PROGRAM PRG_MachineControl
VAR
    // =========================================================
    // TIMERS & TRIGGERS
    // =========================================================
	tonSys_Init           				: TON := (PT := T#8S);    // Initialization pulse timer
    tonSys_InitTimeout    				: TON := (PT := T#15S);   // Initialization timeout fault timer    : TON := (PT := T#15S);   // Initialization timeout fault timer
	tonTimeout_testing    				: TON := (PT := T#20S);   // Initialization timeout fault timer
    tonFirstAutoCycle     				: TON := (PT := T#500MS); // Auto cycle start settling timer
	tonStoppingDelay	  				: TON                   ; // Time to finalize process 
    tonSafety             				: TON := (PT := T#10S);   // Safety interlock debounce timer
	tonAutoCycleIdleTimeout 			: TON := (PT := T#2M);
	tonSimulation		  				: ARRAY[1..4] OF TON; //timer for simulations  
	rtKistlerResultDone   				: R_TRIG;
	rtPartPresentReject   				: R_TRIG;
    
    rtFirstAutoCycle      				: R_TRIG; // Detects entry into Auto Cycle
    fbResetTrigger        				: F_TRIG; // Detects HMI Reset button release
	tTwoHandReturnTimeout 				: TON := (PT := T#2S);
	tonAfterKistlerDelay  				: TON;
	
    eProcessCycleState : E_ProcessCycle_State := E_ProcessCycle_State.IDLE;
	
	tonGuideCylinderDelay 				: TON;
	tonGuideCylinderRetractDelay 		: TON;
	tGuideCylinderDelay   				: TIME := T#250MS;
	
	bFaultResetRequested 				: BOOL := FALSE;
	
    // =========================================================
    // PROCESS CYCLE CONTROL
    // =========================================================
	bStartProcessCondition 				: BOOL;   // OK to Start checklist condition flag
	bAutoCyclePermissive				: BOOL;
    bKistlerReady          				: BOOL;   // Press healthy and ready feedback flag
    i                      				: INT;    // Loop index counter
    sMachineMessage        				: STRING; // Diagnostics and status message string
	stKistlerInTelegram  				: ST_Kistler_TelegramIn;
	stKistlerOutTelegram 				: ST_Kistler_TelegramOut;
	
    bProcessCycleAllowed   		: BOOL;
    bAutoProcessAllowed    		: BOOL;
    bManualKistlerAllowed  		: BOOL;
	
	bAirInitialised     		: BOOL;
	bNestInitialised    		: BOOL;
	bKistlerInitialised 		: BOOL;
	bMachineInitialised 		: BOOL;
	
	bStopRequested 				: BOOL;
	bStopAllowed   				: BOOL;
	
	bRejectConfirmedForExchange : BOOL;
	bPendingOperatorResultPass  : BOOL;
	bPendingOperatorResultFail  : BOOL;
	
	// =================================================================
    // NEST TABLE INTERNAL CONTROL VARIABLES
    // =================================================================
	eNestState           			: E_NestState := E_NestState.IDLE;
	bSequenceToggle      			: BOOL := FALSE;                   // Toggle flag for manual bench testing
	eCurrentNestPos 	 			: E_NestPosition := E_NestPosition.UNKNOWN;
	eCompletedOperatorExchangeNest 	: E_NestPosition;
	
    // HMI PARAMETERS & SAFETY TIMERS
    rHmiTwoHandPresetTime 		: REAL := 250.0; // Time preset from HMI in milliseconds (e.g., 1500.0 ms = 1.5s)
    tTwoHandTargetTime    		: TIME;           // Converted time to be used by the PLC timer
    tTwoHandHoldTimer     		: TON;            // Timer to verify if operator held the buttons long enough
	
	// Timers for pneumatic steps control without sensors
	tSupportRetractDelay 		: TON;  // Time for elevator cylinder to retract down
	tRotatingTableDelay  		: TON;  // Simulated time for index table to complete rotation
	tPortB_ResetDelay    		: TON;  // Pulse time for Port B air relief / mechanism reset
	tSupportExtendDelay  		: TON;  // Time for elevator cylinder to extend back up
	
	eLastTestedNestPos 			: E_NestPosition := E_NestPosition.UNKNOWN;
	bNestNewPositionReady 		: BOOL;

	eOperatorExchangeState : E_OperatorExchangeState := E_OperatorExchangeState.Idle;

	bOperatorExchangeComplete 	 : BOOL;
	bOperatorIndexPermissive   	 : BOOL;
	
	//==========================================================
	//KISTLER COMMAND INTERFACE 
	//==========================================================
	stKistler_CMD          		: ST_Kistler_CMD;    // Commands sent to Kistler press
    stKistler_Status       		: ST_Kistler_Status; // Feedbacks read from Kistler press
	tonKistlerTareYDelay 		: TON;
	
	bKistlerResetPulse  		: BOOL;
    tonKistlerReset     		: TON;
	
	bKistlerRecoveryHomeRequest : BOOL;
	bNestRecoveryHomeRequest	: BOOL;
	uKistlerCurrentValueX 		: U_BytesToReal;
	uKistlerCurrentValueY 		: U_BytesToReal;
	
	// Maximum values recorded during the current Kistler test
	rKistlerCycleMaxForce    	: REAL := 0.0;
	rKistlerCycleMaxDistance 	: REAL := 0.0;

	

	//==========================================================
	//LEDS COMMAND INTERFACE 
	//==========================================================

    // Status memory for each individual LED mode
    eMode_LED_Start    			: E_LEDs_Mode := E_LEDs_Mode.OFF;
    eMode_LED_Reset    			: E_LEDs_Mode := E_LEDs_Mode.OFF;
	eMode_LED_Pass 	   			: E_LEDs_Mode := E_LEDs_Mode.OFF;
    eMode_LED_fail     			: E_LEDs_Mode := E_LEDs_Mode.OFF;
    // Hardware digital outputs mapped to the physical LEDs
    q_bLED_Start      AT%Q*    : BOOL; 
    q_bLED_Reset      AT%Q*    : BOOL;
	q_bLED_Pass       AT%Q*    : BOOL;
	q_bLED_Fail       AT%Q*    : BOOL;
    
	// =========================================================
    // PUCK LOCKER
    // =========================================================
	eKistlerNestPosition  		: E_NestPosition;
    eOperatorNestPosition 		: E_NestPosition;
	ePendingPuckDispositionNest : E_NestPosition := E_NestPosition.Unknown;

    iKistlerNestIndex     		: INT;
    iOperatorNestIndex    		: INT;
	
	bKistlerResultStored 		: BOOL;
	bPartRemovedConfirmedForExchange : BOOL;
	
    // =========================================================
    // PERSISTENT DATA & LOGGING
    // =========================================================
    //fbWritePersistent      : FB_WritePersistentData;
	bWriteTrigger         		: BOOL; // Test and simulation sequence trigger
	eCurrentState				: INT;
	
	// =========================================================
    // HMI COMMAND
    // =========================================================
	bHMIManualModeRequest 		: BOOL := FALSE;
	rtHMIManualModeRequest 		: R_TRIG;
	i_bHMIManualModeRequest		: INT;
	
	
	E_ProcessCycleState			: INT;
	IDLE						: INT;
END_VAR



// =========================================================
// 1. PRE-CONDITION LOGIC
// =========================================================
M_PreExecution();

// Generate Kistler commands based on current machine state
// Map Kistler EtherCAT telegram to PLC status structure
M_KistlerConfig_Output();

bStartProcessCondition :=
    GVL_MASTER.stMachineStatus.bSafety
    AND NOT GVL_MASTER.i_bButtonEmergencyStop
    AND NOT GVL_MASTER.stMachineStatus.bFault
    AND NOT stKistler_Status.bError
    AND stKistler_Status.bReady
    AND GVL_MASTER.stPuckLocker.bMachinePermissive;

 // Initialisation conditions
 
 	
	
    bAirInitialised := GVL_MASTER.bAirSupply_Ok;

    bNestInitialised :=
        (eNestState = E_NestState.IDLE)
        AND NOT GVL_MASTER.stNestTable.bNestInMotion
        AND GVL_MASTER.stNestTable.bNestReadySensor
        AND GVL_MASTER.stNestTable.bNestLockedSensor;

    bKistlerInitialised :=
         stKistler_Status.bInPosition
	      AND NOT stKistler_Status.bError;

    bMachineInitialised :=
        bAirInitialised
        AND bNestInitialised
        AND bKistlerInitialised;
		
	GVL_MASTER.bProcessBusy := 
	(eProcessCycleState <> E_ProcessCycle_State.WAIT_NEST_TESTING_READY 
	AND eProcessCycleState <> E_ProcessCycle_State.IDLE )
	
    OR (eNestState <> E_NestState.IDLE AND eNestState <> E_NestState.FAULT AND eNestState <> E_NestState.WAIT_OPERATOR_EXCHANGE)
    OR GVL_MASTER.stNestTable.bNestInMotion
    OR GVL_MASTER.stProcess.bKistlerCycleRequest
    OR GVL_MASTER.stProcess.bReleaseNestRotation
    OR stKistler_Status.bBusy
    OR NOT stKistler_Status.bInPosition
    OR GVL_MASTER.stNestTable.bSupportExtendRequest
    OR GVL_MASTER.stActuators.bGuideCylinderExtendRequest
	OR GVL_MASTER.stNestTable.bSupportExtended;
	
	

	
// =========================================================
// TIMEOUT
// =========================================================

	tonTimeout_testing (IN := GVL_MASTER.bProcessBusy);
	
	// Any process activity resets the accumulated timeout.
	tonAutoCycleIdleTimeout(
		IN :=
			GVL_MASTER.stMachineStatus.eMachineState =
				E_MachineState.SYSTEM_AUTO_CYCLE
			AND NOT GVL_MASTER.bProcessBusy
	);

// =========================================================
// GLOBAL FAULT DETECTION
// =========================================================
// Only technical Kistler errors shall put the machine in FAULT.
// Kistler NOK result is a rejected part, not a machine fault.
// =========================================================

//OR stKistler_Status.bError
IF (
    NOT GVL_MASTER.stMachineStatus.bSafety
    OR GVL_MASTER.i_bButtonEmergencyStop
)
AND GVL_MASTER.stMachineStatus.eMachineState <> E_MachineState.FAULT THEN

    GVL_MASTER.stMachineStatus.eMachineState := E_MachineState.FAULT;

END_IF;

//HMI Command Manual Mode

rtHMIManualModeRequest(CLK := GVL_HMI.i_bHMIManualModeRequest);

IF rtHMIManualModeRequest.Q AND GVL_Master.stMachineStatus.eMachineState = E_MachineState.SYSTEM_READY_TO_START THEN
    bHMIManualModeRequest := TRUE;
    GVL_HMI.i_bHMIManualModeRequest := FALSE;
ELSE
	bHMIManualModeRequest := FALSE;
    GVL_HMI.i_bHMIManualModeRequest := FALSE;
END_IF;


IF NOT GVL_MASTER.i_bButtonStop THEN
    bStopRequested := TRUE;
END_IF


	
IF GVL_MASTER.stMachineStatus.eMachineState <>
    E_MachineState.FAULT THEN

    bFaultResetRequested := FALSE;
END_IF;
// // =========================================================
// 2. MAIN STATE MACHINE (CASE)
// =========================================================


CASE GVL_Master.stMachineStatus.eMachineState OF


    E_MachineState.SYSTEM_POWER_UP:
	    GVL_Master.stMachineStatus.eMachineState := E_MachineState.STOPPING;
		M_ResetProcessCycle();
		
    E_MachineState.FAULT:
 		eMode_LED_Start := E_LEDs_Mode.OFF;
        eMode_LED_Reset := E_LEDs_Mode.FLASHING; // Reset button must flash
		eMode_LED_Fail := E_LEDs_Mode.ON;
		eMode_LED_PASS := E_LEDs_Mode.OFF;
		
		bHMIManualModeRequest := FALSE;
    	//M_ResetProcessCycle();
		
		 // Store the first reset request while TwinSAFE recovers.
		IF GVL_MASTER.i_bButtonReset THEN
			bFaultResetRequested := TRUE;
		END_IF;

		IF GVL_MASTER.stMachineStatus.bSafety
			AND NOT GVL_MASTER.i_bButtonEmergencyStop
		THEN
			bKistlerResetPulse := TRUE;
		END_IF;
	
	
		IF bKistlerResetPulse THEN
	
			IF M_ResetProcessCycle() THEN
	
				GVL_MASTER.stMachineStatus.eMachineState :=
					E_MachineState.STOPPING;
	
			END_IF;
	
		END_IF;

// 
//         IF  GVL_MASTER.stMachineStatus.bSafety AND NOT GVL_MASTER.i_bButtonEmergencyStop AND fbResetTrigger.Q THEN
//             GVL_Master.stMachineStatus.eMachineState := E_MachineState.STOPPING;
//         END_IF
		
	E_MachineState.STOPPING:
		eMode_LED_PASS := E_LEDs_Mode.OFF;
		eMode_LED_Fail := E_LEDs_Mode.OFF;
        rtFirstAutoCycle(CLK := FALSE);
        tonStoppingDelay(IN := GVL_Master.stMachineStatus.bStopping, PT := T#2S);
		bStopRequested := FALSE;
		IF tonStoppingDelay.Q THEN
			tonStoppingDelay(IN := FALSE);
        	GVL_Master.stMachineStatus.eMachineState := E_MachineState.STOPPED;
		END_IF
	   
	E_MachineState.STOPPED:
		eMode_LED_Reset := E_LEDs_Mode.FLASHING; // Start button must flash
        eMode_LED_Start := E_LEDs_Mode.OFF;
		eMode_LED_PASS := E_LEDs_Mode.OFF;
		eMode_LED_Fail := E_LEDs_Mode.OFF;
		M_ResetProcessCycle();

		IF fbResetTrigger.Q AND bStartProcessCondition THEN
            GVL_Master.stMachineStatus.eMachineState := E_MachineState.SYSTEM_INITIALISING;
			
        END_IF

		
	E_MachineState.SYSTEM_INITIALISING:
	
		tonSys_Init (IN := GVL_MASTER.stMachineStatus.bInitialising);
		tonSys_InitTimeout (IN := GVL_MASTER.stMachineStatus.bInitialising);
		eLastTestedNestPos := E_NestPosition.UNKNOWN;
		
		IF tonSys_Init.Q 
			AND GVL_IO.stSafety.bSafetyOK 
			AND bStartProcessCondition THEN
			
			IF NOT bKistlerInitialised THEN 
				
				 stKistler_Status.eKistlerState := E_KistlerState.HOMING;
    			 bKistlerRecoveryHomeRequest := TRUE;
				
			ELSIF   stKistler_Status.eKistlerState = E_KistlerState.READY THEN
   				GVL_MASTER.stMachineStatus.eMachineState := E_MachineState.SYSTEM_READY_TO_START;
			END_IF
			
		ELSIF tonSys_InitTimeout.Q THEN
			GVL_MASTER.stMachineStatus.eMachineState := E_MachineState.FAULT;
		
		ELSIF bStopRequested THEN
            GVL_Master.stMachineStatus.eMachineState := E_MachineState.STOPPING;
 		END_IF
// 		
	E_MachineState.SYSTEM_READY_TO_START:
	    
		eMode_LED_Start := E_LEDs_Mode.FLASHING; // Start button must flash
        eMode_LED_Reset := E_LEDs_Mode.OFF;
		eMode_LED_PASS := E_LEDs_Mode.OFF;
		eMode_LED_Fail := E_LEDs_Mode.OFF;
		
		IF bStopRequested THEN
            GVL_Master.stMachineStatus.eMachineState := E_MachineState.STOPPING;
	    		
        ELSIF bHMIManualModeRequest
   			AND GVL_MASTER.stMachineStatus.bSafety
   			AND NOT GVL_MASTER.i_bButtonEmergencyStop THEN
			//bHMIManualModeRequest := FALSE;
			GVL_Master.stMachineStatus.eMachineState := E_MachineState.MANUAL_MODE;
			
        ELSIF GVL_MASTER.i_bButtonStart
    			AND bStartProcessCondition
    			AND (stKistler_Status.eKistlerState = E_KistlerState.READY
        		OR stKistler_Status.eKistlerState = E_KistlerState.HOME_DONE) THEN
            		GVL_Master.stMachineStatus.eMachineState := E_MachineState.SYSTEM_AUTO_CYCLE;
			
		ELSIF  NOT GVL_IO.stSafety.bSafetyOK THEN
			GVL_Master.stMachineStatus.eMachineState := E_MachineState.FAULT;
        END_IF	
 
	E_MachineState.SYSTEM_AUTO_CYCLE:
	
		// Show the result of the processed part currently
		// waiting at the operator position.
		// -------------------------------------------------------------------------
		// Operator result indication.
		//
		// The LEDs must represent the stored result of the physical nest currently
		// available to the operator.
		//
		// Do not use bPendingOperatorResultPass / Fail here. Those variables are
		// latched for the operator-exchange state machine and may still represent
		// the previous exchange while the table is indexing.
		// -------------------------------------------------------------------------
		eMode_LED_PASS := E_LEDs_Mode.OFF;
		eMode_LED_Fail := E_LEDs_Mode.OFF;
		
		
		// The operator nest and its array index must be valid.
		IF eOperatorNestPosition <> E_NestPosition.Unknown THEN
		
			iOperatorNestIndex :=
				TO_INT(eOperatorNestPosition);
		
			IF (iOperatorNestIndex >= 1)
			   AND (iOperatorNestIndex <= 4) THEN
		
		
				// -------------------------------------------------------------
				// FAIL indication.
				//
				// Turn the red LED on as soon as the failed part arrives at the
				// operator position.
				//
				// Keep it on after the part is removed from the nest.
				//
				// Turn it off only after the reject sensor confirms that the
				// failed part was placed in the reject location.
				// -------------------------------------------------------------
				IF GVL_MASTER.astNestProcessResult[
						iOperatorNestIndex
				   ].bResultValid
				   AND GVL_MASTER.astNestProcessResult[
						iOperatorNestIndex
				   ].bFail
				   AND NOT bRejectConfirmedForExchange THEN
		
					eMode_LED_PASS := E_LEDs_Mode.OFF;
					eMode_LED_Fail := E_LEDs_Mode.ON;
		
		
				// -------------------------------------------------------------
				// PASS indication.
				//
				// Turn the green LED on as soon as the passed part arrives at
				// the operator position.
				//
				// Turn it off when the operator removes the part from the nest.
				// No puck condition is involved in the indication.
				// -------------------------------------------------------------
				ELSIF GVL_MASTER.astNestProcessResult[
							iOperatorNestIndex
					  ].bResultValid
					  AND GVL_MASTER.astNestProcessResult[
							iOperatorNestIndex
					  ].bPass
					  AND GVL_MASTER.stSensors.bPartPresent_NEST 
					  AND NOT bPartRemovedConfirmedForExchange THEN
		
					eMode_LED_PASS := E_LEDs_Mode.ON;
					eMode_LED_Fail := E_LEDs_Mode.OFF;
		
				END_IF
		
			END_IF
		
		END_IF
	
		rtFirstAutoCycle(CLK := TRUE);
		tonFirstAutoCycle(IN := rtFirstAutoCycle.Q);
	
		IF bStopRequested
			AND NOT GVL_MASTER.bProcessBusy THEN
	
			GVL_MASTER.stMachineStatus.eMachineState :=
				E_MachineState.STOPPING;
	
		ELSIF GVL_MASTER.stMachineStatus.bFault
			OR NOT bStartProcessCondition
			OR NOT GVL_IO.stSafety.bSafetyOK THEN
	
			GVL_MASTER.stMachineStatus.eMachineState :=
				E_MachineState.FAULT;
	
		ELSIF tonTimeout_testing.Q THEN
	
			GVL_MASTER.stMachineStatus.eMachineState :=
				E_MachineState.FAULT;
		ELSIF tonAutoCycleIdleTimeout.Q THEN

			GVL_MASTER.stMachineStatus.eMachineState :=
				E_MachineState.STOPPING;
	
		END_IF;
			
		
		
    E_MachineState.MANUAL_MODE:
		eMode_LED_Start := E_LEDs_Mode.OFF; // Start button must flash
        eMode_LED_Reset := E_LEDs_Mode.OFF;
		eMode_LED_PASS := E_LEDs_Mode.OFF;
		eMode_LED_Fail := E_LEDs_Mode.OFF;
		eLastTestedNestPos := E_NestPosition.UNKNOWN;
   		
		IF NOT GVL_MASTER.stMachineStatus.bSafety
		   OR GVL_MASTER.i_bButtonEmergencyStop THEN
		
			GVL_MASTER.stMachineStatus.eMachineState := E_MachineState.FAULT;
		
		ELSIF  bStopRequested 
			AND NOT GVL_MASTER.bProcessBusy THEN
			GVL_HMI.i_bHMIManualModeRequest				 := FALSE;
    		GVL_HMI.i_bHMIIndexerManualEnable 			 := FALSE;
    		GVL_HMI.i_bHMIKistlerManualEnable 			 := FALSE;
			GVL_MASTER.stMachineStatus.eMachineState := E_MachineState.STOPPING;
		
		END_IF

END_CASE

// =========================================================
// 3. GLOBAL FLAG MAPPING
// =========================================================
GVL_Master.stMachineStatus.bSystemPowerUp := (GVL_Master.stMachineStatus.eMachineState = E_MachineState.SYSTEM_POWER_UP);
GVL_Master.stMachineStatus.bInitialising  := (GVL_Master.stMachineStatus.eMachineState = E_MachineState.SYSTEM_INITIALISING);
GVL_Master.stMachineStatus.bStopped       := (GVL_Master.stMachineStatus.eMachineState = E_MachineState.STOPPED);
GVL_Master.stMachineStatus.bStopping      := (GVL_Master.stMachineStatus.eMachineState = E_MachineState.STOPPING);
GVL_Master.stMachineStatus.bAutoCycle     := (GVL_Master.stMachineStatus.eMachineState = E_MachineState.SYSTEM_AUTO_CYCLE);
GVL_Master.stMachineStatus.bFault         := (GVL_Master.stMachineStatus.eMachineState = E_MachineState.FAULT);
GVL_Master.stMachineStatus.bReadyToStart  := (GVL_Master.stMachineStatus.eMachineState = E_MachineState.SYSTEM_READY_TO_START);
GVL_Master.stMachineStatus.bManualMode    := (GVL_Master.stMachineStatus.eMachineState = E_MachineState.MANUAL_MODE);


// =========================================================
// 5. METHOD POST-EXECUTION ROUTINE
// =========================================================

// Generate base Kistler commands from machine state
M_KistlerControl(
    eCurrentState := GVL_MASTER.stMachineStatus.eMachineState);

// Coordinate Nest and Kistler process sequence
M_ProcessCycle();

// Update Puck locker permissives. 
M_UpdatePuckLockerPermissives();

// Kistler internal state machine may request movement/sequence
M_KistlerStateMachine(
    eCurrentState := GVL_MASTER.stMachineStatus.eMachineState);
	
M_SupportControl(
    bExtendRequest  := GVL_MASTER.stNestTable.bSupportExtendRequest,
    bRetractRequest := GVL_MASTER.stNestTable.bSupportRetractRequest
);

M_GuideCylinderControl(
    bExtendRequest := GVL_MASTER.stActuators.bGuideCylinderExtendRequest
);

M_KistlerConfig_Input();

// Update machine status from Kistler status
M_StatusMapping();

M_LEDsButtons();
M_NestTableControl();

METHOD PRIVATE M_ClearCompletedOperatorNestResult
VAR
	iCompletedNestIndex : INT;
END_VAR
// The nest associated with the completed exchange must be known.
IF eCompletedOperatorExchangeNest = E_NestPosition.Unknown THEN
    RETURN;
END_IF

iCompletedNestIndex := TO_INT(eCompletedOperatorExchangeNest);

IF (iCompletedNestIndex < 1) OR (iCompletedNestIndex > 4) THEN
    RETURN;
END_IF


// Clear only after the complete operator disposition has finished.
GVL_MASTER.astNestProcessResult[iCompletedNestIndex].bResultValid := FALSE;
GVL_MASTER.astNestProcessResult[iCompletedNestIndex].bPass := FALSE;
GVL_MASTER.astNestProcessResult[iCompletedNestIndex].bFail := FALSE;
GVL_MASTER.astNestProcessResult[iCompletedNestIndex].bDispositionSent := FALSE;

eCompletedOperatorExchangeNest := E_NestPosition.Unknown;
END_METHOD

METHOD PRIVATE M_ClearRemovedOperatorNestResult
VAR
	iOperatorNestIndex : INT;
END_VAR
// The operator nest must be known.
IF eOperatorNestPosition = E_NestPosition.Unknown THEN
    RETURN;
END_IF


// E_NestPosition corresponds directly to indexes 1..4.
iOperatorNestIndex := TO_INT(eOperatorNestPosition);

IF (iOperatorNestIndex < 1) OR (iOperatorNestIndex > 4) THEN
    RETURN;
END_IF


// Clear the stored result only when:
//
// 1. The result was already delivered to the Puck Locker.
// 2. The processed part was physically removed from the operator nest.
IF GVL_MASTER.astNestProcessResult[iOperatorNestIndex].bDispositionSent AND GVL_MASTER.astNestTracking[iOperatorNestIndex].bPartRemovedPulse THEN

    GVL_MASTER.astNestProcessResult[iOperatorNestIndex].bResultValid := FALSE;

    GVL_MASTER.astNestProcessResult[iOperatorNestIndex].bPass := FALSE;

    GVL_MASTER.astNestProcessResult[iOperatorNestIndex].bFail := FALSE;

    GVL_MASTER.astNestProcessResult[iOperatorNestIndex].bDispositionSent := FALSE;

END_IF;
END_METHOD

METHOD PRIVATE M_ConfirmPuckLockerDisposition
VAR
	iDispositionNestIndex : INT;
END_VAR
// No disposition is waiting for confirmation.
IF ePendingPuckDispositionNest = E_NestPosition.Unknown THEN
    RETURN;
END_IF


// The Puck Locker has not yet consumed the request.
IF NOT GVL_MASTER.stPuckLocker.bDispositionHandled THEN
    RETURN;
END_IF


// E_NestPosition values correspond directly to indexes 1..4.
iDispositionNestIndex :=
    ePendingPuckDispositionNest;

IF (iDispositionNestIndex < 1) OR (iDispositionNestIndex > 4) THEN

    // Prevent the handshake from remaining blocked by an invalid position.
    ePendingPuckDispositionNest :=
        E_NestPosition.Unknown;
    RETURN;
END_IF


// Mark the result as successfully delivered to the Puck Locker.
GVL_MASTER.astNestProcessResult[iDispositionNestIndex].bDispositionSent := TRUE;


// Release the local handshake.
ePendingPuckDispositionNest := E_NestPosition.Unknown;
END_METHOD

METHOD M_GetCurrentPosition : E_NestPosition
VAR_INST
	iBinaryValue : BYTE;
END_VAR
// 1. Pack the 3 boolean sensors into a single numeric value (Byte) to simplify binary calculation
// Sensor_3 (Bit 2) | Sensor_2 (Bit 1) | Sensor_1 (Bit 0)
iBinaryValue.0 := GVL_MASTER.stNestTable.bNestPos_1_Sensor;
iBinaryValue.1 := GVL_MASTER.stNestTable.bNestPos_2_Sensor;
iBinaryValue.2 := GVL_MASTER.stNestTable.bNestPos_3_Sensor;

// 2. Evaluate the resulting decimal value from the binary combination and return the matching ENUM
CASE iBinaryValue OF
    1: M_GetCurrentPosition := E_NestPosition.POSITION_1; // Binary 001
    2: M_GetCurrentPosition := E_NestPosition.POSITION_2; // Binary 010
    3: M_GetCurrentPosition := E_NestPosition.POSITION_3; // Binary 011
    4: M_GetCurrentPosition := E_NestPosition.POSITION_4; // Binary 100
ELSE
    // Default fallback: If 000 or any unmapped pattern occurs (e.g., 111), the table might be misaligned or in motion
    M_GetCurrentPosition := E_NestPosition.UNKNOWN; 
END_CASE


CASE eCurrentNestPos OF
    E_NestPosition.POSITION_1:
        GVL_HMI.iNestRotationAngle      := 0;
		GVL_HMI.iNestPositionTesting    :=1;

    E_NestPosition.POSITION_2:
        GVL_HMI.iNestRotationAngle 		:= 90;
		GVL_HMI.iNestPositionTesting    :=2;
		
    E_NestPosition.POSITION_3:
        GVL_HMI.iNestRotationAngle 		:= 180;
	    GVL_HMI.iNestPositionTesting    :=3;
		
    E_NestPosition.POSITION_4:
        GVL_HMI.iNestRotationAngle 		:= 270;
		GVL_HMI.iNestPositionTesting    :=4;

ELSE
    GVL_HMI.iNestRotationAngle      := 0;
	GVL_HMI.iNestPositionTesting    := 0;
END_CASE
END_METHOD

METHOD PRIVATE M_GuideCylinderControl
VAR_INPUT
    bExtendRequest : BOOL;
END_VAR
// =================================================================
// GUIDE CYLINDER CONTROL
// =================================================================
// This method is responsible only for the Guide Cylinder output.
// It does not decide Auto Cycle or Manual Mode.
// The request must come from the Kistler state machine.
//
// Single-solenoid pneumatic cylinder:
// TRUE  -> Extend guide cylinder.
// FALSE -> Retract guide cylinder automatically.

GVL_MASTER.stActuators.qGuideCylinder := bExtendRequest;
END_METHOD

METHOD PRIVATE M_HMIKistlerResult : BOOL
VAR_INPUT
    eNestPosition : E_NestPosition;
    bPartOK       : BOOL;
    bPartNOK      : BOOL;
    rForce        : REAL;
    rDistance     : REAL;
	bResetValues  : BOOL;
END_VAR

VAR
    iNestIndex : INT;
END_VAR


M_HMIKistlerResult := FALSE;


// =========================================================
// CONVERT NEST POSITION TO ARRAY INDEX
// =========================================================

CASE eNestPosition OF

    E_NestPosition.Position_1:
        iNestIndex := 1;

    E_NestPosition.Position_2:
        iNestIndex := 2;

    E_NestPosition.Position_3:
        iNestIndex := 3;

    E_NestPosition.Position_4:
        iNestIndex := 4;

ELSE
    RETURN;

END_CASE;


// =========================================================
// RESET VALUES BEFORE A NEW TEST
// =========================================================

IF bResetValues THEN

    GVL_HMI.aKistlerNestResult[iNestIndex].rForce := 0.0;
    GVL_HMI.aKistlerNestResult[iNestIndex].rDistance := 0.0;

    GVL_HMI.aKistlerNestResult[iNestIndex].eResult :=
        E_HMIKistlerResult.NONE;

    M_HMIKistlerResult := TRUE;
    RETURN;

END_IF;


// =========================================================
// STORE MAXIMUM TEST VALUES
// =========================================================

IF ABS(rForce) >
   ABS(GVL_HMI.aKistlerNestResult[iNestIndex].rForce) THEN

    GVL_HMI.aKistlerNestResult[iNestIndex].rForce :=
        rForce;

END_IF;


IF ABS(rDistance) >
   ABS(GVL_HMI.aKistlerNestResult[iNestIndex].rDistance) THEN

    GVL_HMI.aKistlerNestResult[iNestIndex].rDistance :=
        rDistance;

END_IF;


// =========================================================
// STORE FINAL RESULT
// =========================================================

IF bPartOK THEN

    GVL_HMI.aKistlerNestResult[iNestIndex].eResult :=
        E_HMIKistlerResult.PASS;

ELSIF bPartNOK THEN

    GVL_HMI.aKistlerNestResult[iNestIndex].eResult :=
        E_HMIKistlerResult.FAIL;

END_IF;


M_HMIKistlerResult := TRUE;
END_METHOD

METHOD M_IsNestEnabled :BOOL
VAR_INPUT
	   eNestPos : E_NestPosition;
END_VAR
CASE eNestPos OF

    E_NestPosition.Position_1:
        M_IsNestEnabled := GVL_HMI.aNestEnabled[1];

    E_NestPosition.Position_2:
        M_IsNestEnabled := GVL_HMI.aNestEnabled[2];

    E_NestPosition.Position_3:
        M_IsNestEnabled := GVL_HMI.aNestEnabled[3];

    E_NestPosition.Position_4:
        M_IsNestEnabled := GVL_HMI.aNestEnabled[4];

ELSE

    M_IsNestEnabled := FALSE;

END_CASE;
END_METHOD

METHOD PRIVATE M_KistlerCommandMapping : BOOL
VAR
    i : INT;
END_VAR

// =================================================================================
// PLC -> KISTLER COMMAND MAPPING
// =================================================================================
// Clear command telegram
FOR i := 0 TO 199 DO
    GVL_KISTLER_IO.aKistlerOut[i] := 0;
END_FOR

// Enable maXYmos access and automatic mode
IF stKistler_CMD.bEnable THEN
    GVL_KISTLER_IO.aKistlerOut[1].3 := TRUE; // Access
    GVL_KISTLER_IO.aKistlerOut[1].4 := TRUE; // Auto
    GVL_KISTLER_IO.aKistlerOut[9].0 := TRUE; // Drive_Enable
END_IF

// Reset / acknowledge maXYmos faults/statistics
IF stKistler_CMD.bReset THEN
    GVL_KISTLER_IO.aKistlerOut[1].0 := TRUE; // Ack_Admin_Glob
    GVL_KISTLER_IO.aKistlerOut[1].1 := TRUE; // Ack_Admin
    GVL_KISTLER_IO.aKistlerOut[1].5 := TRUE; // Start_Reset
END_IF

// Abort / external sequence stop
IF stKistler_CMD.bAbort THEN
    GVL_KISTLER_IO.aKistlerOut[10].3 := TRUE; // Seq_Ext_Stop
END_IF

// Force Measurement Program 1 for first commissioning test
GVL_KISTLER_IO.aKistlerOut[2].0 := TRUE; // MP_01




M_KistlerCommandMapping := TRUE;
END_METHOD

METHOD PRIVATE M_KistlerConfig_Input : BOOL
VAR
    i : INT;
END_VAR
// =================================================================================
// KISTLER CONFIG INPUT
// PLC -> maXYmos NC input/control telegram
// =================================================================================
// Source:
//     stKistler_CMD
//
// Internal telegram:
//     stKistlerInTelegram
//
// Destination:
//     GVL_KISTLER_IO.aKistlerOut[]
// =================================================================================


// =================================================================================
// CLEAR OUTPUT TELEGRAM
// =================================================================================

FOR i := 0 TO 199 DO
    GVL_KISTLER_IO.aKistlerOut[i] := 0;
END_FOR



// =================================================================================
// HIGH LEVEL COMMANDS -> KISTLER INPUT TELEGRAM STRUCT
// =================================================================================

// -----------------------------------------------------------------------------
// Byte 0 - Measurement commands
// NOTE:
// Byte 0.0 = Measurement START.
// This is NOT the same as Start Sequence.
// Start Sequence is controlled by Byte 9.1 = Run Sequence.
// -----------------------------------------------------------------------------

stKistlerInTelegram.bStart := stKistler_CMD.bStart;
stKistlerInTelegram.bTareY := stKistler_CMD.bTareY;


// -----------------------------------------------------------------------------
// Byte 1 - General control
// -----------------------------------------------------------------------------

stKistlerInTelegram.bAckAdminGlobal := stKistler_CMD.bReset;
stKistlerInTelegram.bAckAdmin       := stKistler_CMD.bReset;
//stKistlerInTelegram.bStatReset      := stKistler_CMD.bReset;
stKistlerInTelegram.bAccess         := stKistler_CMD.bEnable;
stKistlerInTelegram.bAuto           := stKistler_CMD.bEnable;
stKistlerInTelegram.bStatReset       := FALSE;

// -----------------------------------------------------------------------------
// Byte 2 - Measurement program selection
// Byte 2 bits 0..6 = MP selection
// 0 = MP_000
// -----------------------------------------------------------------------------

stKistlerInTelegram.byMeasurementProgram := 0;


// -----------------------------------------------------------------------------
// Byte 9 - Drive / sequence commands
// -----------------------------------------------------------------------------

stKistlerInTelegram.bDriveEnable      := stKistler_CMD.bEnable;
stKistlerInTelegram.bRunSequence      := stKistler_CMD.bRunSequence;
stKistlerInTelegram.bDriveToHomePos   := stKistler_CMD.bDriveToHome;
stKistlerInTelegram.bDriveToRefPos    := stKistler_CMD.bDriveToRef;
stKistlerInTelegram.bContinueFromWait := stKistler_CMD.bContinueFromWait;


// -----------------------------------------------------------------------------
// Byte 10 - External sequence stop request
// -----------------------------------------------------------------------------

stKistlerInTelegram.bSeqExtStopReq := stKistler_CMD.bAbort;


// -----------------------------------------------------------------------------
// Byte 12 - Current sequence selection
// 00 = Main sequence
// 01 = Sub1
// 10 = Sub2
// 11 = Sub3
//
// For current commissioning, always use Main Sequence.
// -----------------------------------------------------------------------------

stKistlerInTelegram.bCurrentSequence0 := FALSE;
stKistlerInTelegram.bCurrentSequence1 := FALSE;


// =================================================================================
// KISTLER INPUT TELEGRAM STRUCT -> OUTPUT BYTES
// =================================================================================

IF stKistlerInTelegram.bDriveToHomePos THEN

    stKistlerInTelegram.bDriveToRefPos := FALSE;
    stKistlerInTelegram.bRunSequence   := FALSE;

ELSIF stKistlerInTelegram.bDriveToRefPos THEN

    stKistlerInTelegram.bDriveToHomePos := FALSE;
    stKistlerInTelegram.bRunSequence    := FALSE;

ELSIF stKistlerInTelegram.bRunSequence THEN

    stKistlerInTelegram.bDriveToHomePos := FALSE;
    stKistlerInTelegram.bDriveToRefPos  := FALSE;

END_IF
// -----------------------------------------------------------------------------
// -----------------------------------------------------------------------------
// Byte 0 - Measurement commands
// Bit 0 = Measurement Start
// Bit 1 = Tare Y
// -----------------------------------------------------------------------------
// -----------------------------------------------------------------------------

GVL_KISTLER_IO.aKistlerOut[0].0 := stKistlerInTelegram.bStart;
GVL_KISTLER_IO.aKistlerOut[0].1 := stKistlerInTelegram.bTareY;


// -----------------------------------------------------------------------------
// Byte 1 - General control
// -----------------------------------------------------------------------------

GVL_KISTLER_IO.aKistlerOut[1].0 := stKistlerInTelegram.bAckAdminGlobal;
GVL_KISTLER_IO.aKistlerOut[1].1 := stKistlerInTelegram.bAckAdmin;
GVL_KISTLER_IO.aKistlerOut[1].3 := stKistlerInTelegram.bAccess;
GVL_KISTLER_IO.aKistlerOut[1].4 := stKistlerInTelegram.bAuto;
GVL_KISTLER_IO.aKistlerOut[1].5 := stKistlerInTelegram.bStatReset;


// -----------------------------------------------------------------------------
// Byte 2 - Measurement program selection
// -----------------------------------------------------------------------------

GVL_KISTLER_IO.aKistlerOut[2] := stKistlerInTelegram.byMeasurementProgram;


// -----------------------------------------------------------------------------
// Byte 9 - Drive / sequence commands
// Bit 0 = Drive Enable
// Bit 1 = Run Sequence / Start Sequence
// Bit 2 = Drive To Home Position
// Bit 3 = Drive To Reference Position
// Bit 6 = Continue From Wait
// -----------------------------------------------------------------------------

GVL_KISTLER_IO.aKistlerOut[9].0 := stKistlerInTelegram.bDriveEnable;
GVL_KISTLER_IO.aKistlerOut[9].1 := stKistlerInTelegram.bRunSequence;
GVL_KISTLER_IO.aKistlerOut[9].2 := stKistlerInTelegram.bDriveToHomePos;
GVL_KISTLER_IO.aKistlerOut[9].3 := stKistlerInTelegram.bDriveToRefPos;
GVL_KISTLER_IO.aKistlerOut[9].6 := stKistlerInTelegram.bContinueFromWait;


// -----------------------------------------------------------------------------
// Byte 10 - External sequence stop request
// Bit 3 = Sequence External Stop Request
// -----------------------------------------------------------------------------

GVL_KISTLER_IO.aKistlerOut[10].3 := stKistlerInTelegram.bSeqExtStopReq;


// -----------------------------------------------------------------------------
// Byte 12 - Current sequence selection
// 00 = Main sequence
// 01 = Sub1
// 10 = Sub2
// 11 = Sub3
// -----------------------------------------------------------------------------

GVL_KISTLER_IO.aKistlerOut[12].0 := stKistlerInTelegram.bCurrentSequence0;
GVL_KISTLER_IO.aKistlerOut[12].1 := stKistlerInTelegram.bCurrentSequence1;


// =================================================================================
// METHOD EXECUTION FEEDBACK
// =================================================================================

M_KistlerConfig_Input := TRUE;
END_METHOD

METHOD PRIVATE M_KistlerConfig_Output : BOOL
VAR_INPUT
END_VAR
// =================================================================================
// INPUT BYTES -> KISTLER OUTPUT TELEGRAM STRUCT
// =================================================================================
// Byte 0 - Mirrored measurement commands
stKistlerOutTelegram.bMirrorStart             := GVL_KISTLER_IO.aKistlerIn[0].0;
stKistlerOutTelegram.bMirrorTareY             := GVL_KISTLER_IO.aKistlerIn[0].1;
stKistlerOutTelegram.bMirrorZeroX             := GVL_KISTLER_IO.aKistlerIn[0].2;
stKistlerOutTelegram.bMirrorSensorTestX       := GVL_KISTLER_IO.aKistlerIn[0].3;
stKistlerOutTelegram.bMirrorSensorTestY       := GVL_KISTLER_IO.aKistlerIn[0].4;
stKistlerOutTelegram.bMirrorMasterMeasurement := GVL_KISTLER_IO.aKistlerIn[0].6;
stKistlerOutTelegram.bMirrorIncZero           := GVL_KISTLER_IO.aKistlerIn[0].7;

// Byte 1 - Mirrored general control
stKistlerOutTelegram.bMirrorAckAdminGlobal := GVL_KISTLER_IO.aKistlerIn[1].0;
stKistlerOutTelegram.bMirrorAckAdmin       := GVL_KISTLER_IO.aKistlerIn[1].1;
stKistlerOutTelegram.bMirrorAccess         := GVL_KISTLER_IO.aKistlerIn[1].3;
stKistlerOutTelegram.bMirrorAuto           := GVL_KISTLER_IO.aKistlerIn[1].4;
stKistlerOutTelegram.bMirrorStatReset      := GVL_KISTLER_IO.aKistlerIn[1].5;
stKistlerOutTelegram.bMirrorStatDisable    := GVL_KISTLER_IO.aKistlerIn[1].6;
stKistlerOutTelegram.bMirrorTareExtendedY  := GVL_KISTLER_IO.aKistlerIn[1].7;

// Byte 2 - Mirrored MP
stKistlerOutTelegram.byMirrorMeasurementProgram := GVL_KISTLER_IO.aKistlerIn[2];

// Byte 3 - Mirrored special commands / reserved
stKistlerOutTelegram.bMirrorResetSNGenerator := GVL_KISTLER_IO.aKistlerIn[3].1;
stKistlerOutTelegram.bMirrorBrakeTestActive  := GVL_KISTLER_IO.aKistlerIn[3].5;
stKistlerOutTelegram.bMirrorExportPVTStatus  := GVL_KISTLER_IO.aKistlerIn[3].6;

// Byte 5 - Reserved
stKistlerOutTelegram.byReserved05 := GVL_KISTLER_IO.aKistlerIn[5];

// Byte 4 - Mirrored configurable inputs
stKistlerOutTelegram.bMirrorInput00 := GVL_KISTLER_IO.aKistlerIn[4].0;
stKistlerOutTelegram.bMirrorInput01 := GVL_KISTLER_IO.aKistlerIn[4].1;
stKistlerOutTelegram.bMirrorInput02 := GVL_KISTLER_IO.aKistlerIn[4].2;
stKistlerOutTelegram.bMirrorInput03 := GVL_KISTLER_IO.aKistlerIn[4].3;
stKistlerOutTelegram.bMirrorInput04 := GVL_KISTLER_IO.aKistlerIn[4].4;
stKistlerOutTelegram.bMirrorInput05 := GVL_KISTLER_IO.aKistlerIn[4].5;
stKistlerOutTelegram.bMirrorInput06 := GVL_KISTLER_IO.aKistlerIn[4].6;
stKistlerOutTelegram.bMirrorInput07 := GVL_KISTLER_IO.aKistlerIn[4].7;

// Byte 6 - General status
stKistlerOutTelegram.bReady    := GVL_KISTLER_IO.aKistlerIn[6].0;
stKistlerOutTelegram.bOkTotal  := GVL_KISTLER_IO.aKistlerIn[6].1;
stKistlerOutTelegram.bNokTotal := GVL_KISTLER_IO.aKistlerIn[6].2;
stKistlerOutTelegram.bWarning  := GVL_KISTLER_IO.aKistlerIn[6].6;
stKistlerOutTelegram.bAlarm    := GVL_KISTLER_IO.aKistlerIn[6].7;

// Byte 9 - Mirrored commands / sequence request
stKistlerOutTelegram.bMirrorDriveEnable    := GVL_KISTLER_IO.aKistlerIn[9].0;
stKistlerOutTelegram.bMirrorRunSequence    := GVL_KISTLER_IO.aKistlerIn[9].1;
stKistlerOutTelegram.bMirrorDriveToHomePos := GVL_KISTLER_IO.aKistlerIn[9].2;
stKistlerOutTelegram.bMirrorDriveToRefPos  := GVL_KISTLER_IO.aKistlerIn[9].3;
stKistlerOutTelegram.bWaitRequest          := GVL_KISTLER_IO.aKistlerIn[9].6;

// Byte 10 - Sequence / drive status
stKistlerOutTelegram.bSequenceStopped := GVL_KISTLER_IO.aKistlerIn[10].0;
stKistlerOutTelegram.bSequenceEnd     := GVL_KISTLER_IO.aKistlerIn[10].1;
//stKistlerOutTelegram.bSequenceError   := GVL_KISTLER_IO.aKistlerIn[10].4;
stKistlerOutTelegram.bSequenceError   := FALSE;
stKistlerOutTelegram.bDriveEnabled    := GVL_KISTLER_IO.aKistlerIn[10].5; // olhar essa 
stKistlerOutTelegram.bHomePosReached  := GVL_KISTLER_IO.aKistlerIn[10].6;
stKistlerOutTelegram.bRefPosReached   := GVL_KISTLER_IO.aKistlerIn[10].7;

// Byte 11 - Servo / safety status
stKistlerOutTelegram.bStandStill       := GVL_KISTLER_IO.aKistlerIn[11].0;
stKistlerOutTelegram.bServoWarning     := GVL_KISTLER_IO.aKistlerIn[11].2;
//stKistlerOutTelegram.bServoError       := GVL_KISTLER_IO.aKistlerIn[11].3;
stKistlerOutTelegram.bServoError       := FALSE;
stKistlerOutTelegram.bSMES_STO         := GVL_KISTLER_IO.aKistlerIn[11].4;
stKistlerOutTelegram.bSMST             := GVL_KISTLER_IO.aKistlerIn[11].5;
stKistlerOutTelegram.bSMM              := GVL_KISTLER_IO.aKistlerIn[11].6;
stKistlerOutTelegram.bUserModeActive   := GVL_KISTLER_IO.aKistlerIn[11].7;

// Byte 19 - Communication status
//stKistlerOutTelegram.bTransmissionFault := GVL_KISTLER_IO.aKistlerIn[19].0;
stKistlerOutTelegram.bTransmissionFault := FALSE;
stKistlerOutTelegram.bAck               := GVL_KISTLER_IO.aKistlerIn[19].1;
stKistlerOutTelegram.bDeviceAvailable   := GVL_KISTLER_IO.aKistlerIn[19].2;

// =================================================================================
// KISTLER OUTPUT TELEGRAM STRUCT -> INTERNAL STATUS
// =================================================================================

// =================================================================================
// INTERNAL STATUS
// =================================================================================

// Kistler is ready from communication/device point of view.
// This does not mean machine is allowed to run.
stKistler_Status.bReady :=
    stKistlerOutTelegram.bDeviceAvailable
    AND NOT stKistlerOutTelegram.bServoError
    AND NOT stKistlerOutTelegram.bTransmissionFault;


// Sequence is running.
// MirrorRunSequence confirms command accepted, and SequenceEnd is still false.
stKistler_Status.bBusy :=
    stKistlerOutTelegram.bMirrorRunSequence
    AND NOT stKistlerOutTelegram.bSequenceEnd
    AND NOT stKistlerOutTelegram.bSequenceStopped;


// Sequence finished, regardless of OK or NOK result.
stKistler_Status.bDone :=
    stKistlerOutTelegram.bSequenceEnd;


// Part result OK.
stKistler_Status.bPartOK :=
    stKistlerOutTelegram.bSequenceEnd
    AND stKistlerOutTelegram.bOkTotal;


// Part result NOK / rejected part.
// Important: this is NOT a technical error.
stKistler_Status.bPartNOK :=
    stKistlerOutTelegram.bSequenceEnd
    AND stKistlerOutTelegram.bNokTotal;


// Technical error only.
// NOK result must not be included here.
// stKistler_Status.bError :=
//     stKistlerOutTelegram.bServoError
//     OR stKistlerOutTelegram.bTransmissionFault
//     OR stKistlerOutTelegram.bSequenceError;


// Position status
stKistler_Status.bInPosition :=
    stKistlerOutTelegram.bHomePosReached;



// =================================================================================
// BYTES 20..23 - CURRENT X VALUE
// X = DISTANCE / DISPLACEMENT / TRAVEL
// =================================================================================

uKistlerCurrentValueX.aBytes[0] := GVL_KISTLER_IO.aKistlerIn[20];
uKistlerCurrentValueX.aBytes[1] := GVL_KISTLER_IO.aKistlerIn[21];
uKistlerCurrentValueX.aBytes[2] := GVL_KISTLER_IO.aKistlerIn[22];
uKistlerCurrentValueX.aBytes[3] := GVL_KISTLER_IO.aKistlerIn[23];

stKistlerOutTelegram.rCurrentValueX :=
    uKistlerCurrentValueX.rValue;


// =================================================================================
// BYTES 24..27 - CURRENT Y VALUE
// Y = FORCE
// =================================================================================

uKistlerCurrentValueY.aBytes[0] := GVL_KISTLER_IO.aKistlerIn[24];
uKistlerCurrentValueY.aBytes[1] := GVL_KISTLER_IO.aKistlerIn[25];
uKistlerCurrentValueY.aBytes[2] := GVL_KISTLER_IO.aKistlerIn[26];
uKistlerCurrentValueY.aBytes[3] := GVL_KISTLER_IO.aKistlerIn[27];

stKistlerOutTelegram.rCurrentValueY :=
    uKistlerCurrentValueY.rValue;
	
	
	// =================================================================================
// MAP LIVE VALUES TO INTERNAL KISTLER STATUS
// =================================================================================

stKistler_Status.rLiveDistance :=
    stKistlerOutTelegram.rCurrentValueX;

stKistler_Status.rLiveForce :=
    stKistlerOutTelegram.rCurrentValueY;


// =================================================================================
// OPTIONAL LIVE VALUES FOR HMI
// =================================================================================

GVL_HMI.rKistlerLiveDistance :=
    stKistler_Status.rLiveDistance;

GVL_HMI.rKistlerLiveForce :=
    stKistler_Status.rLiveForce;
// =================================================================================
// METHOD EXECUTION FEEDBACK
// =================================================================================

M_KistlerConfig_Output := TRUE;
END_METHOD

METHOD PRIVATE M_KistlerControl : BOOL
VAR_INPUT
    eCurrentState : E_MachineState;
END_VAR

VAR
    bKistlerSafetyEnableOK : BOOL;
END_VAR


// =========================================================
// RESET BUTTON DETECTION
// =========================================================

// F_TRIG generates the event when the reset button is released
fbResetTrigger(
    CLK := GVL_MASTER.i_bButtonReset
);


// Perform the complete process reset only in allowed states
IF fbResetTrigger.Q
    AND eCurrentState <> E_MachineState.SYSTEM_AUTO_CYCLE
    AND eCurrentState <> E_MachineState.SYSTEM_READY_TO_START
THEN

    M_ResetProcessCycle();

END_IF;


// =========================================================
// KISTLER RESET / ALARM ACKNOWLEDGEMENT PULSE
// =========================================================

// bKistlerResetPulse is set by M_ResetProcessCycle()
tonKistlerReset(
    IN := bKistlerResetPulse,
    PT := T#500MS
);

// This is the command that is actually sent to the Kistler
stKistler_CMD.bReset := bKistlerResetPulse;


// End the pulse after 500 ms
IF tonKistlerReset.Q THEN

    bKistlerResetPulse := FALSE;

END_IF;


// =========================================================
// ABORT
// =========================================================

// Keep abort active while the machine is faulted
stKistler_CMD.bAbort :=
    eCurrentState = E_MachineState.FAULT;


// =========================================================
// ENABLE
// =========================================================

stKistler_CMD.bEnable :=
    GVL_MASTER.stMachineStatus.bSafety
    AND GVL_KISTLER_IO.bKistlerSafetyEnableOK
    AND NOT GVL_MASTER.i_bButtonEmergencyStop
    AND NOT GVL_MASTER.stMachineStatus.bFault
    AND
    (
        eCurrentState = E_MachineState.SYSTEM_INITIALISING
        OR eCurrentState = E_MachineState.SYSTEM_READY_TO_START
        OR eCurrentState = E_MachineState.SYSTEM_AUTO_CYCLE
        OR eCurrentState = E_MachineState.STOPPING
        OR
        (
            eCurrentState = E_MachineState.MANUAL_MODE
            AND GVL_HMI.i_bHMIKistlerManualEnable
        )
    );


// =========================================================
// MANUAL MODE
// =========================================================

stKistler_CMD.bManualMode :=
    eCurrentState = E_MachineState.MANUAL_MODE
    AND GVL_HMI.i_bHMIKistlerManualEnable;


// =========================================================
// MOTION / SEQUENCE COMMAND DEFAULTS
// =========================================================

// M_KistlerStateMachine(), called later in the PLC cycle,
// may activate these commands when required.

stKistler_CMD.bStart            := FALSE;
stKistler_CMD.bRunSequence      := FALSE;
stKistler_CMD.bDriveToHome      := FALSE;
stKistler_CMD.bDriveToRef       := FALSE;
stKistler_CMD.bContinueFromWait := FALSE;
stKistler_CMD.bTareY            := FALSE;


// =========================================================
// METHOD EXECUTION FEEDBACK
// =========================================================

M_KistlerControl := TRUE;
END_METHOD

METHOD PRIVATE M_KistlerStateMachine : BOOL

VAR_INPUT
    eCurrentState : E_MachineState;

END_VAR

VAR
    bKistlerEnableAllowed    : BOOL;
    bKistlerAutoCycleAllowed : BOOL;
    bKistlerManualAllowed    : BOOL;
    bKistlerSequenceAllowed  : BOOL;
	

	
	
	Teste 			: BOOL :=TRUE;
END_VAR

VAR_INST
    rTrigTwoHands : R_TRIG; // Edge trigger to detect single press of the two-hand safety signal

END_VAR
// =================================================================================
// KISTLER STATE MACHINE
// maXYmos NC logical sequence control
// =================================================================================
// Input:
//     eCurrentState
//     stKistlerOutTelegram
//     stKistler_Status
//
// Output:
//     stKistler_CMD
// =================================================================================


// =================================================================================
// KISTLER OPERATION MODE PERMISSIVES
// =================================================================================

// Kistler may be enabled and stay READY in Ready To Start.
// It may also be enabled during Auto Cycle.
// In Manual Mode, it may be enabled only when the HMI manual enable is active.
bKistlerEnableAllowed :=
    (eCurrentState = E_MachineState.SYSTEM_READY_TO_START)
    OR (eCurrentState = E_MachineState.SYSTEM_AUTO_CYCLE)
	OR (eCurrentState = E_MachineState.SYSTEM_INITIALISING)
    OR (
        (eCurrentState = E_MachineState.MANUAL_MODE)
    );

// Kistler is allowed to run automatically during Auto Cycle.
bKistlerAutoCycleAllowed :=
    (eCurrentState = E_MachineState.SYSTEM_AUTO_CYCLE 
	OR eCurrentState = E_MachineState.SYSTEM_INITIALISING);

// Kistler is allowed to run in Manual Mode only when the HMI manual enable is active.
bKistlerManualAllowed :=
    (eCurrentState = E_MachineState.MANUAL_MODE)
    AND GVL_HMI.i_bHMIKistlerManualEnable;

// Final permissive used by the Kistler sequence.
// Auto Cycle works as before.
// Manual Mode works only when the HMI Kistler manual enable is TRUE.
bKistlerSequenceAllowed :=
    bKistlerAutoCycleAllowed
    OR bKistlerManualAllowed;


// Evaluate positive edge of the safety-certified two-hand control
rTrigTwoHands(CLK := GVL_IO.stSafety.bTwoHandsSafe);
tTwoHandTargetTime := REAL_TO_TIME(rHmiTwoHandPresetTime);   // Convert the HMI float milliseconds value into PLC TIME data type
tTwoHandHoldTimer(IN := GVL_IO.stSafety.bTwoHandsSafe, PT := tTwoHandTargetTime); // Execute the verification timer tied to the physical two-hand safety input





// =================================================================================
// LOCAL / GLOBAL SAFETY AND MACHINE OVERRIDES
// =================================================================================

// Machine stopped, stopping, faulted or Kistler safety not enabled:
// no Kistler movement command is allowed.
IF (eCurrentState = E_MachineState.FAULT)
   OR (eCurrentState = E_MachineState.STOPPING)
   OR (eCurrentState = E_MachineState.STOPPED)
   OR NOT GVL_KISTLER_IO.bKistlerSafetyEnableOK THEN

    stKistler_CMD.bStart := FALSE;              // Byte 0.0 - Measurement Start
    stKistler_CMD.bRunSequence := FALSE;        // Byte 9.1 - Run Sequence
    stKistler_CMD.bDriveToHome := FALSE;        // Byte 9.2 - Drive To Home
    stKistler_CMD.bDriveToRef := FALSE;         // Byte 9.3 - Drive To Reference
    stKistler_CMD.bContinueFromWait := FALSE;   // Byte 9.6 - Continue From Wait
    stKistler_CMD.bTareY := FALSE;              // Byte 0.1 - Tare Y

    stKistler_Status.eKistlerState := E_KistlerState.DISABLED;

    M_KistlerStateMachine := TRUE;
    RETURN;

END_IF;


// Technical Kistler error.
// Important: NOK part result must NOT be treated here as technical error.
// Technical errors are: sequence error, servo error, communication/transmission fault.
IF stKistlerOutTelegram.bSequenceError
   OR stKistlerOutTelegram.bServoError
   OR stKistlerOutTelegram.bTransmissionFault THEN

    stKistler_CMD.bStart := FALSE;
    stKistler_CMD.bRunSequence := FALSE;
    stKistler_CMD.bDriveToHome := FALSE;
    stKistler_CMD.bDriveToRef := FALSE;
    stKistler_CMD.bContinueFromWait := FALSE;
    stKistler_CMD.bTareY := FALSE;

    stKistler_Status.eKistlerState := E_KistlerState.ERROR;
	M_KistlerStateMachine := TRUE;
    RETURN;

END_IF;


// =================================================================================
// ENABLE / READY WITHOUT SEQUENCE
// =================================================================================

// If sequence is not allowed, do not allow Kistler movement commands.
// However, in SYSTEM_READY_TO_START the Kistler can stay enabled and READY.
IF NOT bKistlerSequenceAllowed THEN

    stKistler_CMD.bStart := FALSE;
    stKistler_CMD.bRunSequence := FALSE;
    stKistler_CMD.bDriveToHome := FALSE;
    stKistler_CMD.bDriveToRef := FALSE;
    stKistler_CMD.bContinueFromWait := FALSE;
    stKistler_CMD.bTareY := FALSE;

    // Ready To Start case:
    // Kistler is allowed to be enabled and ready, but no sequence is started.
    IF bKistlerEnableAllowed AND stKistler_CMD.bEnable THEN

        IF stKistler_Status.bError THEN

            stKistler_Status.eKistlerState := E_KistlerState.ERROR;

        ELSE

            IF stKistler_Status.eKistlerState = E_KistlerState.DISABLED THEN
                stKistler_Status.eKistlerState := E_KistlerState.READY;
            END_IF

            IF (stKistler_Status.eKistlerState = E_KistlerState.HOMING)
               OR (stKistler_Status.eKistlerState = E_KistlerState.REFERENCING)
               OR (stKistler_Status.eKistlerState = E_KistlerState.SET_PARAMETERS)
               OR (stKistler_Status.eKistlerState = E_KistlerState.PRESS_READY)
               OR (stKistler_Status.eKistlerState = E_KistlerState.RUN_SEQUENCE)
               OR (stKistler_Status.eKistlerState = E_KistlerState.BUSY) THEN

                stKistler_Status.eKistlerState := E_KistlerState.READY;

            END_IF

        END_IF

    ELSE

        stKistler_Status.eKistlerState := E_KistlerState.DISABLED;

    END_IF

    M_KistlerStateMachine := TRUE;
    RETURN;

END_IF;


// =================================================================================
// KISTLER STATE MACHINE
// =================================================================================

CASE eCurrentState OF

    // =========================================================================
    // AUTO CYCLE OR MANUAL MODE WITH HMI KISTLER ENABLE
    // =========================================================================
    E_MachineState.SYSTEM_AUTO_CYCLE,
	E_MachineState.SYSTEM_INITIALISING,
	E_MachineState.MANUAL_MODE:

        CASE stKistler_Status.eKistlerState OF


            // =========================================================================
            // DISABLED
            // =========================================================================
            E_KistlerState.DISABLED:

                stKistler_CMD.bStart 			:= FALSE;
                stKistler_CMD.bRunSequence 		:= FALSE;
                stKistler_CMD.bDriveToHome 		:= FALSE;
                stKistler_CMD.bDriveToRef 		:= FALSE;
                stKistler_CMD.bContinueFromWait := FALSE;
                stKistler_CMD.bTareY 			:= FALSE;

                IF stKistler_CMD.bEnable THEN
                    stKistler_Status.eKistlerState := E_KistlerState.READY;
                END_IF


            // =========================================================================
            // READY
            // Kistler is enabled and waiting for Auto Cycle or enabled Manual Mode.
            // =========================================================================
            E_KistlerState.READY:

                stKistler_CMD.bStart 			:= FALSE;
                stKistler_CMD.bRunSequence 		:= FALSE;
                stKistler_CMD.bDriveToHome 		:= FALSE;
                stKistler_CMD.bDriveToRef 		:= FALSE;
                stKistler_CMD.bContinueFromWait := FALSE;
                stKistler_CMD.bTareY 			:= FALSE;

                IF stKistler_Status.bError THEN

                    stKistler_Status.eKistlerState := E_KistlerState.ERROR;
					
				ELSIF NOT bKistlerInitialised OR bKistlerRecoveryHomeRequest THEN
					
					stKistler_Status.eKistlerState := E_KistlerState.HOMING;

                ELSIF bKistlerSequenceAllowed
      				AND GVL_MASTER.stProcess.bKistlerCycleRequest THEN

                    // In this project, RefPosReached can be used as initial/home position reference.
                    // If both Home and Ref are false, request homing using DriveToRef.
                    IF NOT stKistlerOutTelegram.bHomePosReached
                       AND NOT stKistlerOutTelegram.bRefPosReached THEN
					   
                        stKistler_Status.eKistlerState := E_KistlerState.HOMING;
	
                    ELSE
						
                        stKistler_Status.eKistlerState := E_KistlerState.SET_PARAMETERS;
						
                    END_IF

               END_IF


            // =========================================================================
            // HOMING
            // Based on reference project TE1096:
            // GOTO_HOME_POS uses DriveToRef command and waits for HomePosReached/RefPosReached.
            // =========================================================================
            E_KistlerState.HOMING:

                stKistler_CMD.bStart 				:= FALSE;
                stKistler_CMD.bRunSequence 			:= FALSE;
                //stKistler_CMD.bDriveToHome 			:= FALSE;
                stKistler_CMD.bContinueFromWait 	:= FALSE;
                stKistler_CMD.bTareY 				:= FALSE;
				
				IF stKistler_CMD.bDriveToRef THEN

    				stKistler_CMD.bDriveToRef := FALSE;

				END_IF;

                // Use DriveToRef for initial/home movement.
                stKistler_CMD.bDriveToRef := TRUE;
				
				IF stKistler_Status.bInPosition 
					AND eCurrentState = E_MachineState.SYSTEM_INITIALISING THEN

    				bKistlerRecoveryHomeRequest := FALSE;
					

				END_IF;

                IF stKistler_Status.bError THEN

                    stKistler_CMD.bDriveToRef := FALSE;
                    stKistler_Status.eKistlerState := E_KistlerState.ERROR;

                ELSIF stKistler_Status.bInPosition 
					OR stKistlerOutTelegram.bHomePosReached
                    OR stKistlerOutTelegram.bRefPosReached THEN

                    stKistler_CMD.bDriveToRef := FALSE;
                    stKistler_Status.eKistlerState := E_KistlerState.HOME_DONE;

                END_IF


            // =========================================================================
            // HOME_DONE
            // Home/reference reached. Next step: prepare parameters.
            // =========================================================================
            E_KistlerState.HOME_DONE:

                stKistler_CMD.bStart := FALSE;
                stKistler_CMD.bRunSequence := FALSE;
                stKistler_CMD.bDriveToHome := FALSE;
                stKistler_CMD.bDriveToRef := FALSE;
                stKistler_CMD.bContinueFromWait := FALSE;
                stKistler_CMD.bTareY := FALSE;

                IF stKistler_Status.bError THEN

                    stKistler_Status.eKistlerState := E_KistlerState.ERROR;

                ELSIF bKistlerSequenceAllowed
     				 AND GVL_MASTER.stProcess.bKistlerCycleRequest THEN

    				stKistler_Status.eKistlerState := E_KistlerState.SET_PARAMETERS;

				ELSE

   					stKistler_Status.eKistlerState := E_KistlerState.READY;

				END_IF


            // =========================================================================
            // SET_PARAMETERS
            // Prepare maXYmos before running sequence.
            // Based on reference project: Tare Y before press cycle.
            // =========================================================================
			E_KistlerState.SET_PARAMETERS:

				stKistler_CMD.bStart := FALSE;
				stKistler_CMD.bRunSequence := FALSE;
				stKistler_CMD.bDriveToHome := FALSE;
				stKistler_CMD.bDriveToRef := FALSE;
				stKistler_CMD.bContinueFromWait := FALSE;
			
				stKistler_CMD.bTareY := TRUE;
			
				tonKistlerTareYDelay(
					IN := stKistlerOutTelegram.bMirrorTareY,
					PT := T#500MS
				);
			
				IF stKistler_Status.bError THEN
			
					stKistler_CMD.bTareY := FALSE;
			
					tonKistlerTareYDelay(IN := FALSE);
					tonGuideCylinderDelay(IN := FALSE);
			
					GVL_MASTER.stActuators.bGuideCylinderExtendRequest := FALSE;
			
					GVL_MASTER.stNestTable.bSupportExtendRequest := FALSE;
					GVL_MASTER.stNestTable.bSupportRetractRequest := TRUE;
			
					stKistler_Status.eKistlerState := E_KistlerState.ERROR;
			
				ELSIF tonKistlerTareYDelay.Q THEN
			
					IF GVL_MASTER.stNestTable.bNestReadySensor
						AND GVL_MASTER.stNestTable.bNestLockedSensor
						AND NOT GVL_MASTER.stNestTable.bNestInMotion
						AND eCurrentNestPos <> E_NestPosition.Unknown THEN
			
						GVL_MASTER.stNestTable.bSupportExtendRequest := TRUE;
						GVL_MASTER.stNestTable.bSupportRetractRequest := FALSE;
			
						IF GVL_MASTER.stNestTable.bSupportExtended THEN
			
							tonGuideCylinderDelay(
								IN := TRUE,
								PT := tGuideCylinderDelay 
							);
			
							IF tonGuideCylinderDelay.Q THEN
			
								GVL_MASTER.stActuators.bGuideCylinderExtendRequest := TRUE;
			
								stKistler_CMD.bTareY := FALSE;
			
								tonKistlerTareYDelay(IN := FALSE);
								tonGuideCylinderDelay(IN := FALSE);
			
								stKistler_Status.eKistlerState := E_KistlerState.PRESS_READY;
			
							ELSE
			
								GVL_MASTER.stActuators.bGuideCylinderExtendRequest := FALSE;
			
							END_IF
			
						ELSE
			
							tonGuideCylinderDelay(IN := FALSE);
							GVL_MASTER.stActuators.bGuideCylinderExtendRequest := FALSE;
			
						END_IF
			
					ELSE
			
						tonGuideCylinderDelay(IN := FALSE);
			
						GVL_MASTER.stActuators.bGuideCylinderExtendRequest := FALSE;
			
						GVL_MASTER.stNestTable.bSupportExtendRequest := FALSE;
						GVL_MASTER.stNestTable.bSupportRetractRequest := TRUE;
			
					END_IF
			
				ELSE
			
					tonGuideCylinderDelay(IN := FALSE);
					GVL_MASTER.stActuators.bGuideCylinderExtendRequest := FALSE;
			
				END_IF
            // =========================================================================
            // PRESS_READY
            // Preparation done. Next step: run sequence.
            // =========================================================================
            E_KistlerState.PRESS_READY:

                tonKistlerTareYDelay(IN := FALSE);

                stKistler_CMD.bStart := FALSE;
                stKistler_CMD.bRunSequence := FALSE;
                stKistler_CMD.bDriveToHome := FALSE;
                stKistler_CMD.bDriveToRef := FALSE;
                stKistler_CMD.bContinueFromWait := FALSE;
                stKistler_CMD.bTareY := FALSE;
				
	
                IF stKistler_Status.bError THEN

                    stKistler_Status.eKistlerState := E_KistlerState.ERROR;

                ELSIF bKistlerSequenceAllowed
      				AND GVL_MASTER.stProcess.bKistlerCycleRequest THEN
					GVL_MASTER.stActuators.bGuideCylinderExtendRequest := TRUE;
					stKistler_Status.eKistlerState := E_KistlerState.RUN_SEQUENCE;
			
				ELSE
			
					stKistler_Status.eKistlerState := E_KistlerState.READY;
			
				END_IF


            // =========================================================================
            // REFERENCING
            // Optional state. Currently not used in normal flow.
            // =========================================================================
            E_KistlerState.REFERENCING:

                stKistler_CMD.bStart := FALSE;
                stKistler_CMD.bRunSequence := FALSE;
                stKistler_CMD.bDriveToHome := FALSE;
                stKistler_CMD.bContinueFromWait := FALSE;
                stKistler_CMD.bTareY := FALSE;

                stKistler_CMD.bDriveToRef := TRUE;

                IF stKistler_Status.bError THEN

                    stKistler_CMD.bDriveToRef := FALSE;
                    stKistler_Status.eKistlerState := E_KistlerState.ERROR;

                ELSIF stKistlerOutTelegram.bRefPosReached THEN

                    stKistler_CMD.bDriveToRef := FALSE;
                    stKistler_Status.eKistlerState := E_KistlerState.REF_DONE;

                END_IF


            // =========================================================================
            // REF_DONE
            // Optional state. Currently not used in normal flow.
            // =========================================================================
            E_KistlerState.REF_DONE:

                stKistler_CMD.bStart := FALSE;
                stKistler_CMD.bRunSequence := FALSE;
                stKistler_CMD.bDriveToHome := FALSE;
                stKistler_CMD.bDriveToRef := FALSE;
                stKistler_CMD.bContinueFromWait := FALSE;
                stKistler_CMD.bTareY := FALSE;

                IF stKistler_Status.bError THEN

                    stKistler_Status.eKistlerState := E_KistlerState.ERROR;

                ELSIF bKistlerSequenceAllowed THEN

                    stKistler_Status.eKistlerState := E_KistlerState.SET_PARAMETERS;

                END_IF


            // =========================================================================
            // RUN_SEQUENCE
            // Command: Start Sequence through RUN-SEQUENCE bit.
            //
            // Important:
            // Byte 9.1 RunSequence = Start Sequence
            // Byte 0.0 Start       = Measurement Start, not sequence start.
            // =========================================================================
			 E_KistlerState.RUN_SEQUENCE:
			
				stKistler_CMD.bStart := FALSE; // Do not use Measurement Start here
				stKistler_CMD.bDriveToHome := FALSE;
				stKistler_CMD.bDriveToRef := FALSE;
				stKistler_CMD.bContinueFromWait := FALSE;
				stKistler_CMD.bTareY := FALSE;
				
				GVL_MASTER.stNestTable.bSupportExtendRequest := TRUE;
				GVL_MASTER.stNestTable.bSupportRetractRequest := FALSE;
				
				GVL_MASTER.stActuators.bGuideCylinderExtendRequest := TRUE;
			
				IF stKistler_Status.bError THEN
			
					stKistler_CMD.bRunSequence := FALSE;
					stKistler_Status.eKistlerState := E_KistlerState.ERROR;
			
				ELSE
			
					// Keep sequence command active until Kistler reacts
					stKistler_CMD.bRunSequence := TRUE;
			
					// If Kistler reports Busy, go to BUSY state
					IF stKistler_Status.bBusy THEN
			
						stKistler_Status.eKistlerState := E_KistlerState.BUSY;
			
					END_IF
			
				END_IF


            // =========================================================================
            // BUSY
            // Sequence is running.
            // Keep RunSequence active during Auto Cycle or enabled Manual Mode.
            // Handle WAIT request if the MP contains WAIT element.
            // =========================================================================
            E_KistlerState.BUSY:

                IF bKistlerSequenceAllowed
   					AND GVL_MASTER.stProcess.bKistlerCycleRequest THEN

				    stKistler_CMD.bStart := FALSE;
					stKistler_CMD.bRunSequence := TRUE;
					stKistler_CMD.bDriveToHome := FALSE;
					stKistler_CMD.bDriveToRef := FALSE;
					stKistler_CMD.bContinueFromWait := FALSE;
					stKistler_CMD.bTareY := FALSE;

                    // Process WAIT handling
                    IF stKistlerOutTelegram.bWaitRequest THEN
                        stKistler_CMD.bContinueFromWait := TRUE;
                    ELSE
                        stKistler_CMD.bContinueFromWait := FALSE;
                    END_IF

                ELSE

                    stKistler_CMD.bRunSequence := FALSE;
                    stKistler_CMD.bDriveToHome := FALSE;
                    stKistler_CMD.bDriveToRef := FALSE;
                    stKistler_CMD.bStart := FALSE;
                    stKistler_CMD.bContinueFromWait := FALSE;
                    stKistler_CMD.bTareY := FALSE;

                    stKistler_Status.eKistlerState := E_KistlerState.READY;

                END_IF

                IF stKistler_Status.bError THEN

                    stKistler_CMD.bRunSequence := FALSE;
                    stKistler_CMD.bDriveToHome := FALSE;
                    stKistler_CMD.bDriveToRef := FALSE;
                    stKistler_CMD.bStart := FALSE;
                    stKistler_CMD.bContinueFromWait := FALSE;
                    stKistler_CMD.bTareY := FALSE;

                    stKistler_Status.eKistlerState := E_KistlerState.ERROR;

                ELSIF stKistlerOutTelegram.bSequenceEnd THEN

                    stKistler_CMD.bRunSequence := FALSE;
                    stKistler_CMD.bDriveToHome := FALSE;
                    stKistler_CMD.bDriveToRef := FALSE;
                    stKistler_CMD.bStart := FALSE;
                    stKistler_CMD.bContinueFromWait := FALSE;
                    stKistler_CMD.bTareY := FALSE;

                    stKistler_Status.eKistlerState := E_KistlerState.DONE;

                ELSIF NOT stKistler_Status.bBusy THEN

                    stKistler_CMD.bContinueFromWait := FALSE;
                    stKistler_CMD.bTareY := FALSE;
                    stKistler_Status.eKistlerState := E_KistlerState.RUN_SEQUENCE;

                END_IF


            // =========================================================================
            // DONE
            // Sequence finished.
            // Result can be OK or NOK.
            // NOK is not a technical error here.
            // =========================================================================
            E_KistlerState.DONE:

				stKistler_CMD.bStart := FALSE;
				stKistler_CMD.bRunSequence := FALSE;
				stKistler_CMD.bDriveToHome := FALSE;
				stKistler_CMD.bDriveToRef := FALSE;
				stKistler_CMD.bContinueFromWait := FALSE;
				stKistler_CMD.bTareY := FALSE;
			
						
				GVL_MASTER.stActuators.bGuideCylinderExtendRequest := FALSE;

				IF stKistler_Status.bError THEN
					tonGuideCylinderRetractDelay(IN := FALSE);
					stKistler_Status.eKistlerState := E_KistlerState.ERROR;
				END_IF
				
				tonGuideCylinderDelay(
					IN := TRUE,
					PT := tGuideCylinderDelay 
				);
				
				IF tonGuideCylinderDelay.Q THEN

					GVL_MASTER.stNestTable.bSupportExtendRequest := FALSE;
					GVL_MASTER.stNestTable.bSupportRetractRequest := TRUE;
				
					IF NOT GVL_MASTER.stProcess.bKistlerCycleRequest
						AND NOT GVL_MASTER.stProcess.bNestTestingReady
						AND NOT GVL_MASTER.stProcess.bReleaseNestRotation THEN
				
						tonGuideCylinderRetractDelay(IN := FALSE);
				
						IF stKistler_CMD.bEnable THEN
								stKistler_Status.eKistlerState := E_KistlerState.READY;
						ELSE
								stKistler_Status.eKistlerState := E_KistlerState.DISABLED;
						END_IF
				
					END_IF
				
				END_IF

            // =========================================================================
            // ERROR
            // Technical error state.
            // Commands are disabled until error clears and reset/enable condition returns.
            // =========================================================================
            E_KistlerState.ERROR:

                stKistler_CMD.bStart := FALSE;
                stKistler_CMD.bRunSequence := FALSE;
                stKistler_CMD.bDriveToHome := FALSE;
                stKistler_CMD.bDriveToRef := FALSE;
                stKistler_CMD.bContinueFromWait := FALSE;
                stKistler_CMD.bTareY := FALSE;
				
				GVL_MASTER.stNestTable.bSupportExtendRequest  := FALSE;
				GVL_MASTER.stNestTable.bSupportRetractRequest := TRUE;

                IF NOT stKistler_Status.bError THEN

                    IF stKistler_CMD.bEnable THEN
                        stKistler_Status.eKistlerState := E_KistlerState.READY;
                    ELSE
                        stKistler_Status.eKistlerState := E_KistlerState.DISABLED;
                    END_IF

                END_IF

        END_CASE;



    // =========================================================================
    // MACHINE FAULT
    // =========================================================================
    E_MachineState.FAULT:

        stKistler_CMD.bStart 							:= FALSE;
        stKistler_CMD.bRunSequence 						:= FALSE;
        stKistler_CMD.bDriveToHome 						:= FALSE;
        stKistler_CMD.bDriveToRef 						:= FALSE;
        stKistler_CMD.bContinueFromWait 				:= FALSE;
        stKistler_CMD.bTareY 							:= FALSE;
		GVL_MASTER.stNestTable.bSupportExtendRequest  	:= FALSE;
		GVL_MASTER.stNestTable.bSupportRetractRequest 	:= TRUE;

        IF stKistler_Status.eKistlerState <> E_KistlerState.DISABLED THEN
            stKistler_Status.eKistlerState := E_KistlerState.ERROR;
        END_IF


    // =========================================================================
    // OTHER MACHINE STATES
    // =========================================================================
		ELSE
	
			stKistler_CMD.bStart 			:= FALSE;
			stKistler_CMD.bRunSequence 		:= FALSE;
			stKistler_CMD.bDriveToHome 		:= FALSE;
			stKistler_CMD.bDriveToRef 		:= FALSE;
			stKistler_CMD.bContinueFromWait := FALSE;
			stKistler_CMD.bTareY 			:= FALSE;

END_CASE;

// =================================================================================
// METHOD EXECUTION FEEDBACK
// =================================================================================

M_KistlerStateMachine := TRUE;
END_METHOD

METHOD M_LEDsButtons : BOOL
VAR_INST
    // Static-like variables inside the method (Instantiated with the PRG)
    fbBlinker         : TON;
    bBlinkerPulse     : BOOL;
END_VAR
// =================================================================
// 1. INTERNAL BLINKER GENERATOR
// =================================================================
fbBlinker(IN := NOT fbBlinker.Q, PT := T#500MS);
IF fbBlinker.Q THEN
    bBlinkerPulse := NOT bBlinkerPulse;
END_IF;

// =================================================================
// 2. PROCESS START LED HARDWARE OUTPUT
// =================================================================
CASE PRG_MachineControl.eMode_LED_Start OF
    E_LEDs_Mode.ON:
        PRG_MachineControl.q_bLED_Start := TRUE;
        
    E_LEDs_Mode.FLASHING:
        PRG_MachineControl.q_bLED_Start := bBlinkerPulse;
        
    E_LEDs_Mode.OFF:
        PRG_MachineControl.q_bLED_Start := FALSE;
END_CASE;

// =================================================================
// 3. PROCESS RESET LED HARDWARE OUTPUT
// =================================================================
CASE PRG_MachineControl.eMode_LED_Reset OF
    E_LEDs_Mode.ON:
        PRG_MachineControl.q_bLED_Reset := TRUE;
        
    E_LEDs_Mode.FLASHING:
        PRG_MachineControl.q_bLED_Reset := bBlinkerPulse;
        
    E_LEDs_Mode.OFF:
        PRG_MachineControl.q_bLED_Reset := FALSE;
END_CASE;
// =================================================================
// 4. PROCESS LED PASS HARDWARE OUTPUT
// =================================================================
CASE PRG_MachineControl.eMode_LED_Pass OF
    E_LEDs_Mode.ON:
        PRG_MachineControl.q_bLED_Pass := TRUE;
        
    E_LEDs_Mode.FLASHING:
        PRG_MachineControl.q_bLED_Pass := bBlinkerPulse;
        
    E_LEDs_Mode.OFF:
        PRG_MachineControl.q_bLED_Pass := FALSE;
END_CASE;

// =================================================================
// 4. PROCESS LED FAIL HARDWARE OUTPUT
// =================================================================
CASE PRG_MachineControl.eMode_LED_Fail OF
    E_LEDs_Mode.ON:
        PRG_MachineControl.q_bLED_Fail := TRUE;
        
    E_LEDs_Mode.FLASHING:
        PRG_MachineControl.q_bLED_Fail := bBlinkerPulse;
        
    E_LEDs_Mode.OFF:
        PRG_MachineControl.q_bLED_Fail := FALSE;
END_CASE;



M_LEDsButtons := TRUE;
END_METHOD

METHOD M_NestTableControl
VAR_INST
    rTrigTwoHands 				: R_TRIG; // Edge trigger to detect single press of the two-hand safety signal
	
	bNestAutoCycleAllowed 		: BOOL;
	bNestManualAllowed    		: BOOL;
	bNestSequenceAllowed  		: BOOL;
	
END_VAR

// =================================================================
// STATE PERMISSIONS
// =================================================================

bNestAutoCycleAllowed := GVL_MASTER.stMachineStatus.eMachineState = E_MachineState.SYSTEM_AUTO_CYCLE;

bNestManualAllowed := GVL_MASTER.stMachineStatus.eMachineState = E_MachineState.MANUAL_MODE AND GVL_HMI.i_bHMIIndexerManualEnable;

bNestSequenceAllowed := bNestAutoCycleAllowed OR bNestManualAllowed;

// =================================================================
// Puck Locker fault interlock.
//
// Only automatic production depends on the Puck Locker.
//
// In Manual Mode, the machine must behave exactly as before the
// Puck Locker feature existed.
// =================================================================
IF GVL_MASTER.stMachineStatus.eMachineState =
    E_MachineState.SYSTEM_AUTO_CYCLE THEN

    IF GVL_MASTER.stPuckLocker.bUnexpectedRemovalFault
       OR GVL_MASTER.stPuckLocker.bPuckSensorMismatch
       OR GVL_MASTER.stPuckLocker.eState =
            E_PuckLockerState.UnexpectedPuckRemovalFault THEN

        GVL_MASTER.stNestTable.qNestRotatePortA := FALSE;
        GVL_MASTER.stNestTable.qNestRotatePortB := FALSE;
        GVL_MASTER.stNestTable.bNestInMotion    := FALSE;

        GVL_MASTER.stProcess.bNestTestingReady     := FALSE;
        GVL_MASTER.stProcess.bReleaseNestRotation  := FALSE;

        eNestState := E_NestState.FAULT;

        RETURN;

    END_IF

END_IF


IF NOT bNestSequenceAllowed
   AND GVL_MASTER.stMachineStatus.eMachineState <>
       E_MachineState.FAULT THEN

    GVL_MASTER.stNestTable.qNestRotatePortA := FALSE;
    GVL_MASTER.stNestTable.qNestRotatePortB := FALSE;
    GVL_MASTER.stNestTable.bNestInMotion 	:= FALSE;
    GVL_MASTER.stProcess.bNestTestingReady 	:= FALSE;

    eNestState := E_NestState.IDLE;
    RETURN;

END_IF

// =================================================================
// 1. EMERGENCY RESET AND GLOBAL INTERLOCK PROCESSING
// =================================================================
// Global asynchronous reset: Forces the system to IDLE and drops all outputs immediately
IF fbResetTrigger.Q 
	AND NOT GVL_Master.stMachineStatus.bAutoCycle
	AND NOT GVL_Master.stMachineStatus.bReadyToStart THEN
	
    eNestState                              		:= E_NestState.IDLE;
    bSequenceToggle                         		:= FALSE; // Always restart from rotation step after reset
    GVL_MASTER.stNestTable.bNestStartCycle  		:= FALSE;
    GVL_MASTER.stNestTable.bNestInMotion    		:= FALSE;
    GVL_MASTER.stNestTable.qNestRotatePortA 		:= FALSE;
    GVL_MASTER.stNestTable.qNestRotatePortB 		:= FALSE;
    GVL_MASTER.stNestTable.bSupportExtendRequest    := FALSE;
    GVL_MASTER.stNestTable.bSupportRetractRequest   := TRUE;  // Safe home posture for elevator

    RETURN; // Abort remaining logic execution for this cycle
END_IF

// Global Safety Interlock: Force fault state immediately if air/safety is lost
IF NOT GVL_IO.stSafety.bSafetyOK AND GVL_Master.stMachineStatus.bFault THEN
    eNestState := E_NestState.FAULT;
END_IF

//eCurrentNestPos := M_GetCurrentPosition();

// =================================================================
// 2. INPUT SIGNAL PROCESSING (TRIGGERS)
// =================================================================
// Evaluate positive edge of the safety-certified two-hand control
rTrigTwoHands(CLK := GVL_IO.stSafety.bTwoHandsSafe);
tTwoHandTargetTime := REAL_TO_TIME(rHmiTwoHandPresetTime);   // Convert the HMI float milliseconds value into PLC TIME data type
tTwoHandHoldTimer(IN := GVL_IO.stSafety.bTwoHandsSafe, PT := tTwoHandTargetTime); // Execute the verification timer tied to the physical two-hand safety input

// Trigger processing to allow automated cycle start from IDLE state
// IF rTrigTwoHands.Q AND GVL_MASTER.bStations_Home AND GVL_IO.stSafety.bSafetyOK AND (eNestState = E_NestState.IDLE) THEN
//      IF GVL_MASTER.stMachineStatus.bAutoCycle THEN
//          GVL_MASTER.stNestTable.bNestInMotion := TRUE;
//          eNestState                           := E_NestState.ROTATING_TABLE; // Start the automated cycle directly at rotation step
//      END_IF
// END_IF

// =================================================================
// 3. TIMERS EXECUTION (CYCLIC COUPLING TO MAIN PROGRAM INSTANCES)
// =================================================================
// Enchained timers execution pattern to generate an automated timeline for the TESTING state
tRotatingTableDelay(IN  := (eNestState = E_NestState.ROTATING_TABLE), PT := T#500MS);
tPortB_ResetDelay(IN    := (eNestState = E_NestState.STOP_TABLE), PT := T#1S);

// TESTING TIMELINE: 
// 1. Initial 100ms settling delay starts when entering TESTING state
tSupportRetractDelay(IN := (eNestState = E_NestState.TESTING), PT := T#100MS);
// 2. 2-Second lift holding duration executes after the initial pause finishes
tSupportExtendDelay(IN  := (eNestState = E_NestState.TESTING) AND tSupportRetractDelay.Q, PT := T#200MS);

// Two-hand return timeout.
// If the operator does not press the two-hand control again within 1 second,
// the sequence goes to FAULT.
tTwoHandReturnTimeout(IN := (eNestState = E_NestState.WRONG_POSITION),PT := T#5S);

// =================================================================
// 4. NEST TABLE STATE MACHINE CONTROL (WITH INTERNAL INTERLOCKS)
// =================================================================
CASE GVL_Master.stMachineStatus.eMachineState OF    
    
    E_MachineState.SYSTEM_AUTO_CYCLE,
	E_MachineState.MANUAL_MODE:
        
        CASE eNestState OF
        
            E_NestState.IDLE:

				GVL_MASTER.stNestTable.qNestRotatePortA := FALSE;
				GVL_MASTER.stNestTable.qNestRotatePortB := FALSE;
				GVL_MASTER.stNestTable.bNestInMotion    := FALSE;
				GVL_MASTER.stProcess.bNestTestingReady  := FALSE;
			//
				IF GVL_IO.stSafety.bSafetyOK
				   AND rTrigTwoHands.Q
				   AND GVL_MASTER.bStations_Home
				   AND GVL_MASTER.stNestTable.bSupportRetracted
				   AND bNestSequenceAllowed
				   AND (
						GVL_MASTER.stMachineStatus.eMachineState =
							E_MachineState.MANUAL_MODE
						OR
						GVL_MASTER.stPuckLocker.bIndexPermissive
					)
				   AND stKistler_Status.bInPosition
				   AND NOT stKistler_Status.bBusy THEN
				
					GVL_MASTER.stNestTable.bNestInMotion := TRUE;
					eNestState := E_NestState.ROTATING_TABLE;
				
				END_IF
        
            E_NestState.ROTATING_TABLE: // State 2: ROTATING TABLE

				GVL_MASTER.stNestTable.bNestInMotion      := TRUE;
				GVL_MASTER.stProcess.bNestTestingReady    := FALSE;
				GVL_MASTER.stNestTable.bSupportExtendRequest := FALSE;
			    GVL_MASTER.stNestTable.bSupportRetractRequest := TRUE;
			
				IF NOT GVL_IO.stSafety.bSafetyOK THEN
			
					GVL_MASTER.stNestTable.qNestRotatePortA := FALSE;
					GVL_MASTER.stNestTable.qNestRotatePortB := FALSE;
					eNestState := E_NestState.FAULT;
			
				ELSIF NOT GVL_IO.stSafety.bTwoHandsSafe
					  AND NOT tTwoHandHoldTimer.Q THEN
			
					GVL_MASTER.stNestTable.qNestRotatePortA := FALSE;
					GVL_MASTER.stNestTable.qNestRotatePortB := FALSE;
					eNestState := E_NestState.WRONG_POSITION;
			
				ELSIF NOT bNestSequenceAllowed THEN
			
					GVL_MASTER.stNestTable.qNestRotatePortA := FALSE;
					GVL_MASTER.stNestTable.qNestRotatePortB := FALSE;
					eNestState := E_NestState.IDLE;
			
				ELSIF GVL_MASTER.stNestTable.bSupportRetracted 
					AND NOT stKistler_Status.bBusy 
					AND NOT GVL_MASTER.stActuators.bGuideCylinderExtendRequest
					AND stKistler_Status.bInPosition
					AND NOT GVL_MASTER.stProcess.bKistlerCycleRequest THEN
			
					GVL_MASTER.stNestTable.qNestRotatePortA := TRUE;
					GVL_MASTER.stNestTable.qNestRotatePortB := FALSE;
			
					IF tRotatingTableDelay.Q
					   AND GVL_MASTER.stNestTable.bNestCompletedSensor THEN
			
						eNestState := E_NestState.STOP_TABLE;
			
					END_IF
			
				ELSE
					// Support is not retracted. Do not rotate.
					GVL_MASTER.stNestTable.qNestRotatePortA := FALSE;
					GVL_MASTER.stNestTable.qNestRotatePortB := FALSE;
			
				END_IF
        
            E_NestState.STOP_TABLE: // State 3: STOP TABLE

				GVL_MASTER.stProcess.bNestTestingReady := FALSE;
			
				GVL_MASTER.stNestTable.qNestRotatePortA := FALSE;
				GVL_MASTER.stNestTable.qNestRotatePortB := TRUE;
			
				IF NOT GVL_IO.stSafety.bSafetyOK THEN
			
					GVL_MASTER.stNestTable.qNestRotatePortA := FALSE;
					GVL_MASTER.stNestTable.qNestRotatePortB := FALSE;
					eNestState := E_NestState.FAULT;
			
				ELSIF NOT bNestSequenceAllowed THEN
			
					GVL_MASTER.stNestTable.qNestRotatePortA := FALSE;
					GVL_MASTER.stNestTable.qNestRotatePortB := FALSE;
					GVL_MASTER.stNestTable.bNestInMotion    := FALSE;
					eNestState := E_NestState.IDLE;
			
				ELSIF tPortB_ResetDelay.Q
					  AND GVL_MASTER.stNestTable.bNestReadySensor
					  AND GVL_MASTER.stNestTable.bNestLockedSensor THEN
			
					GVL_MASTER.stNestTable.bNestInMotion    := FALSE;
					GVL_MASTER.stNestTable.qNestRotatePortB := FALSE;
					eNestState := E_NestState.TESTING;
			
				END_IF
        
			E_NestState.TESTING: // State 4: TESTING / Kistler test position
			
				GVL_MASTER.stNestTable.qNestRotatePortA := FALSE;
				GVL_MASTER.stNestTable.qNestRotatePortB := FALSE;
				GVL_MASTER.stNestTable.bNestInMotion := FALSE;
			
			
				IF NOT GVL_IO.stSafety.bSafetyOK THEN
			
					GVL_MASTER.stProcess.bNestTestingReady := FALSE;
					eNestState := E_NestState.FAULT;
			
			
				ELSIF NOT bNestSequenceAllowed THEN
			
					GVL_MASTER.stProcess.bNestTestingReady := FALSE;
					eNestState := E_NestState.IDLE;
			
			
				ELSIF NOT GVL_MASTER.stNestTable.bNestReadySensor
					  OR NOT GVL_MASTER.stNestTable.bNestLockedSensor
					  OR eCurrentNestPos = E_NestPosition.Unknown THEN
			
					GVL_MASTER.stProcess.bNestTestingReady := FALSE;
					eNestState := E_NestState.FAULT;
			
			
				ELSE
			
					// Table is stopped and safely positioned for the Kistler process.
					GVL_MASTER.stProcess.bNestTestingReady := TRUE;
			
			
					// The Process Cycle has completed the Kistler operation
					// and is requesting the nest to leave the testing phase.
					IF GVL_MASTER.stProcess.bReleaseNestRotation THEN
			
						GVL_MASTER.stProcess.bNestTestingReady := FALSE;
						GVL_MASTER.stProcess.bReleaseNestRotation := FALSE;
			
						// Do not rotate yet. First wait for the operator exchange.
						eNestState := E_NestState.WAIT_OPERATOR_EXCHANGE;
			
					END_IF
			
				END_IF
				
			E_NestState.WAIT_OPERATOR_EXCHANGE:

				// The Kistler test is finished.
				// Keep the table stationary while the operator completes:
				// - processed-part removal;
				// - puck exchange when required;
				// - new puck locking;
				// - new-part loading.
			
				GVL_MASTER.stNestTable.qNestRotatePortA := FALSE;
				GVL_MASTER.stNestTable.qNestRotatePortB := FALSE;
				GVL_MASTER.stNestTable.bNestInMotion 	:= FALSE;
			
				GVL_MASTER.stProcess.bNestTestingReady 		:= FALSE;
				GVL_MASTER.stProcess.bReleaseNestRotation 	:= FALSE;
			
			
				IF NOT GVL_IO.stSafety.bSafetyOK THEN
			
					eNestState := E_NestState.FAULT;
			
			
				ELSIF NOT bNestSequenceAllowed THEN
			
					eNestState := E_NestState.IDLE;
			
			
				ELSIF NOT GVL_MASTER.stNestTable.bNestReadySensor
					  OR NOT GVL_MASTER.stNestTable.bNestLockedSensor
					  OR eCurrentNestPos = E_NestPosition.Unknown THEN
			
					eNestState := E_NestState.FAULT;
			
			
				ELSIF     (
					GVL_MASTER.stMachineStatus.eMachineState =
						E_MachineState.MANUAL_MODE
					OR
					GVL_MASTER.stPuckLocker.bIndexPermissive
				) THEN
			
					// Operator exchange completed.
					// Return to IDLE, where the existing two-hand logic
					// can start the next pneumatic index.
					eNestState := E_NestState.IDLE;
			
				END_IF
			
				
				
			E_NestState.WRONG_POSITION: // State 99: WRONG_POSITION (Emergency Stop or Air Loss)

				GVL_MASTER.stNestTable.qNestRotatePortA := FALSE;
				GVL_MASTER.stNestTable.qNestRotatePortB := TRUE;
				GVL_MASTER.stNestTable.bNestInMotion    := TRUE;
			
				GVL_MASTER.stProcess.bNestTestingReady  := FALSE;
			
				IF tTwoHandReturnTimeout.Q THEN
			
					GVL_MASTER.stNestTable.qNestRotatePortA := FALSE;
					GVL_MASTER.stNestTable.qNestRotatePortB := FALSE;
					GVL_MASTER.stNestTable.bNestInMotion    := FALSE;
			
					eNestState := E_NestState.FAULT;
			
				ELSIF rTrigTwoHands.Q
					  AND GVL_IO.stSafety.bSafetyOK
					  AND bNestSequenceAllowed
					  AND GVL_MASTER.stNestTable.bSupportRetracted THEN
			
					GVL_MASTER.stNestTable.qNestRotatePortA := TRUE;
					GVL_MASTER.stNestTable.qNestRotatePortB := FALSE;
			
					eNestState := E_NestState.ROTATING_TABLE;
			
				ELSIF GVL_IO.stSafety.bSafetyOK
					  AND NOT GVL_MASTER.stMachineStatus.bFault
					  AND GVL_MASTER.stNestTable.bNestReadySensor
					  AND eCurrentNestPos <> E_NestPosition.Unknown THEN
			
					GVL_MASTER.stNestTable.qNestRotatePortA := FALSE;
					GVL_MASTER.stNestTable.qNestRotatePortB := FALSE;
					GVL_MASTER.stNestTable.bNestInMotion    := FALSE;
			
					eNestState := E_NestState.STOP_TABLE;
			
				END_IF
				
            E_NestState.FAULT:

					GVL_MASTER.stNestTable.qNestRotatePortA := FALSE;
					GVL_MASTER.stNestTable.qNestRotatePortB := FALSE;
					GVL_MASTER.stNestTable.bNestInMotion    := FALSE;
				
					GVL_MASTER.stProcess.bNestTestingReady  := FALSE;
					GVL_MASTER.stProcess.bReleaseNestRotation := FALSE;
				
					GVL_MASTER.stNestTable.bSupportExtendRequest  := FALSE;
					GVL_MASTER.stNestTable.bSupportRetractRequest := TRUE;
				
					GVL_MASTER.stMachineStatus.eMachineState := E_MachineState.FAULT;

        END_CASE

    // =================================================================
    // FAULT 
    // =================================================================
	
	E_MachineState.FAULT:
	
	 				GVL_MASTER.stNestTable.qNestRotatePortA := FALSE;
					GVL_MASTER.stNestTable.qNestRotatePortB := FALSE;
					GVL_MASTER.stNestTable.bNestInMotion    := FALSE;
				
					GVL_MASTER.stProcess.bNestTestingReady  := FALSE;
					GVL_MASTER.stProcess.bReleaseNestRotation := FALSE;
				
					GVL_MASTER.stNestTable.bSupportExtendRequest  := FALSE;
					GVL_MASTER.stNestTable.bSupportRetractRequest := TRUE;

	    IF GVL_IO.stSafety.bSafetyOK AND NOT GVL_Master.stMachineStatus.bFault THEN
        	eNestState := E_NestState.IDLE;
        END_IF

	

		
	END_CASE
END_METHOD

METHOD PRIVATE M_OperatorExchangeControl
VAR
	iOperatorNestIndex 	: INT;
    bOperatorResultPass : BOOL;
    bOperatorResultFail : BOOL;
	bOperatorResultValid : BOOL;
END_VAR
// Default value prevents stale index permission.
bOperatorExchangeComplete := FALSE;


// -----------------------------------------------------------------------------
// Validate the nest currently accessible to the operator.
// -----------------------------------------------------------------------------
IF eOperatorNestPosition = E_NestPosition.Unknown THEN
    RETURN;
END_IF


iOperatorNestIndex := TO_INT(eOperatorNestPosition);

IF (iOperatorNestIndex < 1) OR (iOperatorNestIndex > 4) THEN
    RETURN;
END_IF


// -----------------------------------------------------------------------------
// Result associated with the nest currently accessible to the operator.
// -----------------------------------------------------------------------------
bOperatorResultValid :=
    GVL_MASTER.astNestProcessResult[
        iOperatorNestIndex
    ].bResultValid;


bOperatorResultPass :=
    GVL_MASTER.astNestProcessResult[
        iOperatorNestIndex
    ].bResultValid
    AND
    GVL_MASTER.astNestProcessResult[
        iOperatorNestIndex
    ].bPass;


bOperatorResultFail :=
    GVL_MASTER.astNestProcessResult[
        iOperatorNestIndex
    ].bResultValid
    AND
    GVL_MASTER.astNestProcessResult[
        iOperatorNestIndex
    ].bFail;

// -----------------------------------------------------------------------------
// Retain operator actions even while the Kistler is processing another nest.
//
// Both the nest removal pulse and the reject sensor pulse last only one PLC
// scan. They must therefore be retained immediately and not only when the
// exchange state machine reaches the corresponding waiting state.
// -----------------------------------------------------------------------------

// A processed part was removed from the operator nest.
IF (
        bOperatorResultValid
        OR bPendingOperatorResultPass
        OR bPendingOperatorResultFail
   )
   AND GVL_MASTER.astNestTracking[
        iOperatorNestIndex
   ].bPartRemovedPulse THEN

    bPartRemovedConfirmedForExchange := TRUE;

END_IF


// A failed part was placed at the reject sensor.
IF (
        bOperatorResultFail
        OR bPendingOperatorResultFail
   )
   AND rtPartPresentReject.Q THEN

    bRejectConfirmedForExchange := TRUE;

END_IF


// ============================================================================
// Operator exchange sequence
// ============================================================================
CASE eOperatorExchangeState OF


    // ========================================================================
    E_OperatorExchangeState.Idle:
    // ========================================================================

        bOperatorExchangeComplete := FALSE;

        // Preserve the physical nest associated with this exchange.
        eCompletedOperatorExchangeNest :=
            eOperatorNestPosition;


        // --------------------------------------------------------------------
        // Case 1:
        // A tested result is pending at the operator nest.
        //
        // The processed part must be handled before the table may index.
        // --------------------------------------------------------------------
        IF
			(
				(
					eNestState = E_NestState.IDLE
					OR
					eNestState = E_NestState.WAIT_OPERATOR_EXCHANGE
					OR
					(
						eNestState = E_NestState.TESTING
						AND bOperatorResultPass
					)
				)
				AND NOT GVL_MASTER.stNestTable.bNestInMotion
				AND GVL_MASTER.stNestTable.bNestReadySensor
				AND GVL_MASTER.stNestTable.bNestLockedSensor
				AND bOperatorResultValid
			)
			THEN

            // Latch the result for the entire operator exchange.
            //
            // Do not reset these variables every PLC cycle.
            bPendingOperatorResultPass :=
                bOperatorResultPass;

            bPendingOperatorResultFail :=
                bOperatorResultFail;

           //bRejectConfirmedForExchange := FALSE;


			// -------------------------------------------------------------
			// The processed part may already have been removed while another
			// nest was being tested.
			//
			// If the operator already loaded a new part, the physical sensor
			// will be ON again. Therefore, the retained removal event must
			// take priority over the current sensor state.
			// -------------------------------------------------------------
			IF bPartRemovedConfirmedForExchange THEN
			
				// ---------------------------------------------------------
				// PASS result.
				// ---------------------------------------------------------
				IF bOperatorResultPass THEN
			
					IF GVL_HMI.stPuckLocker.eMode =
						E_PuckLockerMode.Disabled THEN
			
						eOperatorExchangeState :=
							E_OperatorExchangeState.ExchangeComplete;
			
					ELSE
			
						eOperatorExchangeState :=
							E_OperatorExchangeState.WaitingForPuckRemoval;
			
					END_IF
			
			
				// ---------------------------------------------------------
				// FAIL result.
				// ---------------------------------------------------------
				ELSIF bOperatorResultFail THEN
			
					eOperatorExchangeState :=
						E_OperatorExchangeState.WaitingForRejectConfirmation;
			
				END_IF
			
			
			// -------------------------------------------------------------
			// No removal event was retained and the processed part is still
			// physically present.
			//
			// Wait for the operator to remove it.
			// -------------------------------------------------------------
			ELSIF GVL_MASTER.stSensors.bPartPresent_NEST THEN
			
				eOperatorExchangeState :=
					E_OperatorExchangeState.WaitingForPartRemoval;
			
			
			// -------------------------------------------------------------
			// The part is already absent, for example after fault recovery
			// or machine restart.
			// -------------------------------------------------------------
			ELSE
			
				bPartRemovedConfirmedForExchange := TRUE;
			
				// ---------------------------------------------------------
				// PASS result.
				// ---------------------------------------------------------
				IF bOperatorResultPass THEN
			
					IF GVL_HMI.stPuckLocker.eMode =
						E_PuckLockerMode.Disabled THEN
			
						eOperatorExchangeState :=
							E_OperatorExchangeState.ExchangeComplete;
			
					ELSE
			
						eOperatorExchangeState :=
							E_OperatorExchangeState.WaitingForPuckRemoval;
			
					END_IF
			
			
				// ---------------------------------------------------------
				// FAIL result.
				// ---------------------------------------------------------
				ELSIF bOperatorResultFail THEN
			
					eOperatorExchangeState :=
						E_OperatorExchangeState.WaitingForRejectConfirmation;
			
				END_IF
			
			END_IF


        // --------------------------------------------------------------------
        // Case 2:
        // No tested result is pending.
        //
        // Enabled:
        //     Require a present and locked puck.
        //
        // Disabled:
        //     Ignore only the physical puck conditions.
        // --------------------------------------------------------------------
        ELSIF (
                eNestState = E_NestState.IDLE
                OR
                eNestState = E_NestState.WAIT_OPERATOR_EXCHANGE
              )
              AND NOT GVL_MASTER.stNestTable.bNestInMotion
              AND GVL_MASTER.stNestTable.bNestReadySensor
              AND GVL_MASTER.stNestTable.bNestLockedSensor
              AND NOT bOperatorResultValid
              AND (
                    GVL_HMI.stPuckLocker.eMode =
                        E_PuckLockerMode.Disabled

                    OR
                    (
                        GVL_MASTER.stPuckLocker.bPuckDetected
                        AND
                        GVL_MASTER.stPuckLocker.bPuckLocked
                        AND
                        GVL_MASTER.stPuckLocker.eState =
                            E_PuckLockerState.Locked
                    )
              ) THEN

            bPendingOperatorResultPass := FALSE;
            bPendingOperatorResultFail := FALSE;

            bPartRemovedConfirmedForExchange := FALSE;
            bRejectConfirmedForExchange := FALSE;

            eOperatorExchangeState :=
                E_OperatorExchangeState.ExchangeComplete;

        END_IF


    // ========================================================================
    E_OperatorExchangeState.WaitingForPartRemoval:
    // ========================================================================

        bOperatorExchangeComplete := FALSE;


        // This state is entered only when a processed part was confirmed
        // present in the operator nest.
        //
        // Therefore, the part has been removed when the physical sensor
        // becomes FALSE.
        IF bPartRemovedConfirmedForExchange
   			OR NOT GVL_MASTER.stSensors.bPartPresent_NEST THEN

            bPartRemovedConfirmedForExchange := TRUE;


            // -------------------------------------------------------------
            // PASS result.
            // -------------------------------------------------------------
            IF bPendingOperatorResultPass THEN

                // With the Puck Locker disabled, removal of the good part
                // completes the operator exchange.
                IF GVL_HMI.stPuckLocker.eMode =
                    E_PuckLockerMode.Disabled THEN

